(* IEC 61131-3 sources: SJ_AGV/PLC (part 2) *)

   END_STRUCT;
END_TYPE
TYPE
    LanSerialPort_T :
    STRUCT
        Protocol : DINT ;   (* Protocol used for IP communication.  *)
        IP : STRING ;   (* In case of Protocol set to UDP client or TCP client this should be set
to the IP address of the UDP/TCP server that the PLC connects to. With
Protocol set to UDP server or TCP server this specify the IP address of
the vehicle controller which clients should use.

In the case of Protocol set to UDP server or TCP server, the special
value "LAN" means that connections are only allowed on the
LAN interface and the special value "ANY" allows connections
on both the LAN interface and the WLAN interface.

Changing the address from the PLC will result in the connection being
closed. The new IP address will be used in the next PLC loop serial
read/write.  Note! It is not possible to change the address for a
range sensor connected using a LAN-serial-adapter.  *)
        Port : DINT ;   (* In case of Protocol set to UDP client or TCP client this should be set
to the port of the UDP/TCP server that the PLC connects to. With
Protocol set to UDP server or TCP server this specify the port on the
vehicle controller that the PLC opens for connections.

Changing the port from the PLC will result in the connection being
closed. The new port will be used in the next PLC loop serial
read/write.  Note! It is not possible to change the port for a range
sensor connected using a LAN-serial-adapter.  *)
        SendBuffer : BOOL ;   (* With SendBuffer set, outgoing data is sent over IP when the PLC
function block NDC_SERIAL_WRITE is called with argument
LENGTH=0. Without SendBuffer set, data is sent immediately but each IP
packet will contain at most 32 bytes data with more IP traffic as a
result.  *)

   END_STRUCT;
END_TYPE
TYPE
    UserDefined_T :
    STRUCT
        DoNavInit : BOOL ;   (* Boolean_1  *)
        Braker_Signal : BOOL ;   (* Boolean_2  *)
        DoLocalOrder : BOOL ;   (* Boolean_3  *)
        ChangeOrderMode : BOOL ;   (* Boolean_4  *)
        LowBatSim : BOOL ;   (* Boolean_5  *)
        Boolean_6 : BOOL ;   (* Boolean_6  *)
        Boolean_7 : BOOL ;   (* Boolean_7  *)
        Boolean_8 : BOOL ;   (* Boolean_8  *)
        Boolean_9 : BOOL ;   (* Boolean_9  *)
        Boolean_10_BlockPowOffEn : BOOL ;   (* Boolean_10  *)
        Boolean_11_LostPosPowOffEn : BOOL ;   (*   *)
        Boolean_12 : BOOL ;   (*   *)
        Boolean_13 : BOOL ;   (*   *)
        Boolean_14 : BOOL ;   (*   *)
        Boolean_15 : BOOL ;   (*   *)
        Boolean_16 : BOOL ;   (*   *)
        Boolean_17 : BOOL ;   (*   *)
        Boolean_18 : BOOL ;   (*   *)
        Boolean_19 : BOOL ;   (*   *)
        Boolean_20_OnlineOrderMode : BOOL ;   (* 1 = Local Mode; 0 = Host Mode  *)
        Boolean_21 : BOOL ;   (*   *)
        Boolean_22 : BOOL ;   (*   *)
        Boolean_23 : BOOL ;   (*   *)
        Boolean_24 : BOOL ;   (*   *)
        Boolean_25 : BOOL ;   (*   *)
        Boolean_26 : BOOL ;   (*   *)
        Boolean_27 : BOOL ;   (*   *)
        Boolean_28 : BOOL ;   (*   *)
        Boolean_29 : BOOL ;   (*   *)
        Boolean_30 : BOOL ;   (*   *)
        StopWord : DINT ;   (* Integer32_1  *)
        Integer32_2 : DINT ;   (* Integer32_2  *)
        Integer32_3 : DINT ;   (* Integer32_3  *)
        Integer32_4 : DINT ;   (* Integer32_4  *)
        Integer32_5 : DINT ;   (* Integer32_5  *)
        SlowDownDisable : DINT ;   (* Integer32_6  *)
        PPAEnable : DINT ;   (* Integer32_7  *)
        SafetyScannerTurnAngle : DINT ;   (* Integer32_8  *)
        NormalCreepDistance : DINT ;   (* Integer32_9  *)
        Integer32_10 : DINT ;   (* Integer32_10  *)
        Integer32_11 : DINT ;   (* Integer32_11  *)
        Integer32_12 : DINT ;   (* Integer32_12  *)
        Integer32_13 : DINT ;   (* Integer32_13  *)
        Integer32_14 : DINT ;   (* Integer32_14  *)
        Integer32_15 : DINT ;   (* Integer32_15  *)
        Integer32_16 : DINT ;   (* Integer32_16  *)
        Integer32_17 : DINT ;   (* Integer32_17  *)
        Integer32_18 : DINT ;   (* Integer32_18  *)
        Integer32_19 : DINT ;   (* Integer32_19  *)
        Integer32_20 : DINT ;   (* Integer32_20  *)
        Integer32_21 : DINT ;   (* Integer32_21  *)
        Integer32_22 : DINT ;   (* Integer32_22  *)
        Integer32_23 : DINT ;   (* Integer32_23  *)
        Integer32_24 : DINT ;   (* Integer32_24  *)
        Integer32_25 : DINT ;   (* Integer32_25  *)
        Integer32_26 : DINT ;   (* Integer32_26  *)
        Integer32_27 : DINT ;   (* Integer32_27  *)
        Integer32_28 : DINT ;   (* Integer32_28  *)
        Integer32_29 : DINT ;   (* Integer32_29  *)
        Integer32_30 : DINT ;   (* Integer32_30  *)
        Integer32_31 : DINT ;   (* Integer32_31  *)
        Integer32_32 : DINT ;   (* Integer32_32  *)
        Integer32_33 : DINT ;   (* Integer32_33  *)
        Integer32_34 : DINT ;   (* Integer32_34  *)
        Integer32_35 : DINT ;   (* Integer32_35  *)
        Integer32_36 : DINT ;   (* Integer32_36  *)
        Integer32_37 : DINT ;   (* Integer32_37  *)
        Integer32_38 : DINT ;   (* Integer32_38  *)
        Integer32_39 : DINT ;   (* Integer32_39  *)
        Integer32_40 : DINT ;   (* Integer32_40  *)
        Integer32_41 : DINT ;   (* Integer32_41  *)
        Integer32_42 : DINT ;   (* Integer32_42  *)
        Integer32_43 : DINT ;   (* Integer32_43  *)
        Integer32_44 : DINT ;   (* Integer32_44  *)
        Integer32_45 : DINT ;   (* Integer32_45  *)
        Integer32_46 : DINT ;   (* Integer32_46  *)
        Integer32_47 : DINT ;   (*   *)
        Integer32_48 : DINT ;   (*   *)
        Integer32_49 : DINT ;   (*   *)
        Integer32_50_BattLowVol : DINT ;   (*   *)
        Integer32_51_BattLowSel : DINT ;   (* 1=L or M or H, 2=M or H, 3=H  *)
        Integer32_52_PowOffTm : DINT ;   (* ms  *)
        Integer32_53 : DINT ;   (*   *)
        Integer32_54 : DINT ;   (*   *)
        Integer32_55_TravelDistance : DINT ;   (*   *)
        Integer32_56 : DINT ;   (*   *)
        Integer32_57 : DINT ;   (*   *)
        Integer32_58_LS2000_Attached_D : DINT ;   (*   *)
        Integer32_59_LS2000_Attached_H : DINT ;   (*   *)
        Integer32_60_LS2000_Attached_M : DINT ;   (*   *)

   END_STRUCT;
END_TYPE
TYPE
    SDIO_T :
    STRUCT
        IMUGyroX : INT ;   (* Gyroscope x-axis value, cdeg/s  *)
        IMUGyroY : INT ;   (* Gyroscope y-axis value, cdeg/s  *)
        IMUGyroZ : INT ;   (* Gyroscope z-axis value, cdeg/s  *)
        IMUAccX : INT ;   (* Accelerometer x-axis value, mg  *)
        IMUAccY : INT ;   (* Accelerometer x-axis value, mg  *)
        IMUAccZ : INT ;   (* Accelerometer x-axis value, mg  *)
        IMUError : UINT ;   (* IMU Error value  *)
        IMUGyroXScale : INT ;   (* Gyroscope x-axis scale value (the value 10000 corresponds to a real scale value of 1.0)  *)
        IMUGyroYScale : INT ;   (* Gyroscope y-axis scale value (the value 10000 corresponds to a real scale value of 1.0)  *)
        IMUGyroZScale : INT ;   (* Gyroscope z-axis scale value (the value 10000 corresponds to a real scale value of 1.0)  *)
        DigitalInput1_Polarity : BOOL ;   (* Digital Input 1 Polarity, pin #A22  *)
        DigitalInput2_Polarity : BOOL ;   (* Digital Input 2 Polarity, pin #A14  *)
        DigitalInput3_Polarity : BOOL ;   (* Digital Input 3 Polarity, pin #A7  *)
        DigitalInput4_Polarity : BOOL ;   (* Digital Input 4 Polarity, pin #A6  *)
        DigitalInput5_Polarity : BOOL ;   (* Digital Input 5 Polarity, pin #A13  *)
        DigitalInput6_Polarity : BOOL ;   (* Digital Input 6 Polarity, pin #A21  *)
        DigitalInput7_Polarity : BOOL ;   (* Digital Input 7 Polarity, pin #A20  *)
        DigitalInput8_Polarity : BOOL ;   (* Digital Input 8 Polarity, pin #A19  *)
        DigitalInput9_Polarity : BOOL ;   (* Digital Input 9 Polarity, pin #B22  *)
        DigitalInput10_Polarity : BOOL ;   (* Digital Input 10 Polarity, pin #B23  *)
        DigitalInput11_Polarity : BOOL ;   (* Digital Input 11 Polarity, pin #A18  *)
        DigitalInput12_Polarity : BOOL ;   (* Digital Input 12 Polarity, pin #A17  *)
        DigitalOutput2_Polarity : BOOL ;   (* Digital Output 2 Polarity, pin #B7  *)
        DigitalOutput3_Polarity : BOOL ;   (* Digital Output 3 Polarity, pin #B6  *)
        DigitalOutput4_Polarity : BOOL ;   (* Digital Output 4 Polarity, pin #B5  *)
        DigitalOutput5_Polarity : BOOL ;   (* Digital Output 5 Polarity, pin #B4  *)
        DigitalOutput6_Polarity : BOOL ;   (* Digital Output 6 Polarity, pin #B1  *)
        DigitalOutput7_Polarity : BOOL ;   (* Digital Output 7 Polarity, pin #B3  *)
        DigitalOutput8_Polarity : BOOL ;   (* Digital Output 8 Polarity, pin #B2  *)
        DigitalOutput12_Polarity : BOOL ;   (* Digital Output 12 Polarity, pin #A3  *)
        DigitalOutput13_Polarity : BOOL ;   (* Digital Output 13 Polarity, pin #A10  *)
        DigitalOutput14_Polarity : BOOL ;   (* Digital Output 14 Polarity, pin #A2  *)
        DigitalOutput15_Polarity : BOOL ;   (* Digital Output 15 Polarity, pin #A9  *)
        DigitalOutput16_Polarity : BOOL ;   (* Digital Output 16 Polarity, pin #A16  *)
        AnInp1_Scale : DINT ;   (* Analog Input 1 Scale, pin #B15  *)
        AnInp2_Scale : DINT ;   (* Analog Input 2 Scale, pin #B17  *)
        AnInp3_Scale : DINT ;   (* Analog Input 3 Scale, pin #B10  *)
        AnInp4_Scale : DINT ;   (* Analog Input 4 Scale, pin #B18  *)
        AnInp5_Scale : DINT ;   (* Analog Input 5 Scale, pin #B11  *)
        AnInp6_Scale : DINT ;   (* Analog Input 6 Scale, pin #B19  *)
        AnInp7_Scale : DINT ;   (* Analog Input 7 Scale, pin #B12  *)
        AnInp8_Scale : DINT ;   (* Analog Input 8 Scale, pin #B20  *)
        AnInp9_Scale : DINT ;   (* Analog Input 9 Scale, pin #B13  *)
        AnInp10_Scale : DINT ;   (* Analog Input 10 Scale, pin #B21  *)
        AnInp11_Scale : DINT ;   (* Analog Input 11 Scale, pin #B14  *)
        AnInp1_Delta : UDINT ;   (* Asynchroneous transmission will be triggered if input has changed more than this value since last transmission.  *)
        AnInp2_Delta : UDINT ;   (* Asynchroneous transmission will be triggered if input has changed more than this value since last transmission.  *)
        AnInp3_Delta : UDINT ;   (* Asynchroneous transmission will be triggered if input has changed more than this value since last transmission.  *)
        AnInp4_Delta : UDINT ;   (* Asynchroneous transmission will be triggered if input has changed more than this value since last transmission.  *)
        AnInp5_Delta : UDINT ;   (* Asynchroneous transmission will be triggered if input has changed more than this value since last transmission.  *)
        AnInp6_Delta : UDINT ;   (* Asynchroneous transmission will be triggered if input has changed more than this value since last transmission.  *)
        AnInp7_Delta : UDINT ;   (* Asynchroneous transmission will be triggered if input has changed more than this value since last transmission.  *)
        AnInp8_Delta : UDINT ;   (* Asynchroneous transmission will be triggered if input has changed more than this value since last transmission.  *)
        AnInp9_Delta : UDINT ;   (* Asynchroneous transmission will be triggered if input has changed more than this value since last transmission.  *)
        AnInp10_Delta : UDINT ;   (* Asynchroneous transmission will be triggered if input has changed more than this value since last transmission.  *)
        AnInp11_Delta : UDINT ;   (* Asynchroneous transmission will be triggered if input has changed more than this value since last transmission.  *)
        AnInp1_Offset : DINT ;   (* Analog Input 1 Offset, pin #B15  *)
        AnInp2_Offset : DINT ;   (* Analog Input 2 Offset, pin #B17  *)
        AnInp3_Offset : DINT ;   (* Analog Input 3 Offset, pin #B10  *)
        AnInp4_Offset : DINT ;   (* Analog Input 4 Offset, pin #B18  *)
        AnInp5_Offset : DINT ;   (* Analog Input 5 Offset, pin #B11  *)
        AnInp6_Offset : DINT ;   (* Analog Input 6 Offset, pin #B19  *)
        AnInp7_Offset : DINT ;   (* Analog Input 7 Offset, pin #B12  *)
        AnInp8_Offset : DINT ;   (* Analog Input 8 Offset, pin #B20  *)
        AnInp9_Offset : DINT ;   (* Analog Input 9 Offset, pin #B13  *)
        AnInp10_Offset : DINT ;   (* Analog Input 10 Offset, pin #B21  *)
        AnInp11_Offset : DINT ;   (* Analog Input 11 Offset, pin #B14  *)
        DigitalInput1_BTN_STR : BOOL ;   (* Digital Input 1 value, pin #A22  *)
        DigitalInput2_BTN_RST : BOOL ;   (* Digital Input 2 value, pin #A14  *)
        DigitalInput3_BMP_O1 : BOOL ;   (* Digital Input 3 value, pin #A7  *)
        DigitalInput4_BMP_O2 : BOOL ;   (* Digital Input 4 value, pin #A6  *)
        DigitalInput5_BTN_BRK : BOOL ;   (* Digital Input 5 value, pin #A13  *)
        DigitalInput6 : BOOL ;   (* Digital Input 6 value, pin #A21  *)
        DigitalInput7 : BOOL ;   (* Digital Input 7 value, pin #A20  *)
        DigitalInput8_BMP_E : BOOL ;   (* Digital Input 8 value, pin #A19  *)
        DigitalInput9 : BOOL ;   (* Digital Input 9 value, pin #B22  *)
        DigitalInput10 : BOOL ;   (* Digital Input 10 value, pin #B23  *)
        DigitalInput11 : BOOL ;   (* Digital Input 11 value, pin #A18  *)
        DigitalInput12_EMO : BOOL ;   (* Digital Input 12 value, pin #A17  *)
        AllOK_DigitalOutput1 : BOOL ;   (* Reserved Digital Output 1 (All-OK, pin #B8)  *)
        DigitalOutput2_LEDF_L : BOOL ;   (* Digital Output 2 value, pin #B7  *)
        DigitalOutput3_LEDF_R : BOOL ;   (* Digital Output 3 value, pin #B6  *)
        DigitalOutput4_LEDR_L : BOOL ;   (* Digital Output 4 value, pin #B5  *)
        DigitalOutput5_LEDR_R : BOOL ;   (* Digital Output 5 value, pin #B4  *)
        DigitalOutput6_LED_INPOS : BOOL ;   (* Digital Output 6 value, pin #B1  *)
        DigitalOutput7_LED_STR : BOOL ;   (* Digital Output 7 value, pin #B3  *)
        DigitalOutput8_LED_RST : BOOL ;   (* Digital Output 8 value, pin #B2  *)
        DigitalOutput12 : BOOL ;   (* Digital Output 12 value, pin #A3  *)
        DigitalOutput13_PWR_OFF : BOOL ;   (* Digital Output 13 value, pin #A10  *)
        DigitalOutput14_LED_BRK : BOOL ;   (* Digital Output 14 value, pin #A2  *)
        DigitalOutput15 : BOOL ;   (* Digital Output 15 value, pin #A9  *)
        DigitalOutput16_Charger : BOOL ;   (* Digital Output 16 value, pin #A16  *)
        AnalogInput1 : INT ;   (* Analog Input 1 value, pin #B15. The value is the applied input voltage (in Volts) * Scale + Offset  *)
        AnalogInput2 : INT ;   (* Analog Input 2 value, pin #B17. The value is the applied input voltage (in Volts) * Scale + Offset  *)
        AnalogInput3 : INT ;   (* Analog Input 3 value, pin #B10. The value is the applied input voltage (in Volts) * Scale + Offset  *)
        AnalogInput4 : INT ;   (* Analog Input 4 value, pin #B18. The value is the applied input voltage (in Volts) * Scale + Offset  *)
        AnalogInput5 : INT ;   (* Analog Input 5 value, pin #B11. The value is the applied input voltage (in Volts) * Scale + Offset  *)
        AnalogInput6 : INT ;   (* Analog Input 6 value, pin #B19. The value is the applied input voltage (in Volts) * Scale + Offset  *)
        AnalogInput7 : INT ;   (* Analog Input 7 value, pin #B12. The value is the applied input voltage (in Volts) * Scale + Offset  *)
        AnalogInput8 : INT ;   (* Analog Input 8 value, pin #B20. The value is the applied input voltage (in Volts) * Scale + Offset  *)
        AnalogInput9 : INT ;   (* Analog Input 9 value, pin #B13. The value is the applied input voltage (in Volts) * Scale + Offset  *)
        AnalogInput10 : INT ;   (* Analog Input 10 value, pin #B21. The value is the applied input voltage (in Volts) * Scale + Offset  *)
        AnalogInput11 : INT ;   (* Analog Input 11 value, pin #B14. The value is the applied input voltage (in Volts) * Scale + Offset  *)
        PWMOutput1 : INT ;   (* PWM Output 1 value, pin #A5. The value is the duty cycle of the output.  *)
        PWMOutput2 : INT ;   (* PWM Output 2 value, pin #A12. The value is the duty cycle of the output.  *)
        PWMOutput3 : INT ;   (* PWM Output 3 value, pin #A11. The value is the duty cycle of the output.  *)
        Reg1Output : INT ;   (* Regulator 1 output value  *)
        Reg2Output : INT ;   (* Regulator 2 output value  *)
        GroundFaultEvent : BOOL ;   (* If set to true, a ground fault will cause a system event 229.  *)
        GroundFaultActive : BOOL ;   (* True if a ground fault is present  *)
        Temperature : DINT ;   (* Current temperature  *)
        XV_Out : DINT ;   (* Current xv out voltage  *)
        B_Plus : DINT ;   (* Current b plus voltage  *)
        BusID : DINT ;   (* CAN bus ID  *)
        NodeID : DINT ;   (* CAN node ID  *)
        FailureAction : DINT ;   (* 0 = Background, the background programs takes action when an error occur in the device. 1 = PLC, no action from background program. The error should be handled by the PLC application.  *)
        ActiveInSafeState : BOOL ;   (* Decides if the device will start up in safe state.  *)
        NMTState : UDINT ;   (* The current CANopen state of the device.  *)
        SdoBufferSize : DINT ;   (* The current size of the client SDO buffer (read/write SDO's from the vehicle controller to this device).  *)
        IMUAxis : STRING ;   (* The axis in the IMU that gives the angular rate for vehicle.  *)
        IMUNavActive : BOOL ;   (* Use the angular rate from the IMU when calculating the position of the vehicle.  *)

   END_STRUCT;
END_TYPE
TYPE
    CAN_IO_3_T :
    STRUCT
        DigitalInput1_SteerLimitF_L : BOOL ;   (* Digital Input 1 value  *)
        DigitalInput2_SteerLimitF_R : BOOL ;   (* Digital Input 2 value  *)
        DigitalInput3_SteerLimitR_L : BOOL ;   (* Digital Input 3 value  *)
        DigitalInput4_SteerLimitR_R : BOOL ;   (* Digital Input 4 value  *)
        DigitalInput5_LIMF_O : BOOL ;   (* Digital Input 5 value  *)
        DigitalInput6_LIMR_O : BOOL ;   (* Digital Input 6 value  *)
        DigitalInput7 : BOOL ;   (* Digital Input 7 value  *)
        DigitalInput8 : BOOL ;   (* Digital Input 8 value  *)
        DigitalInput9_AreaF_IN1 : BOOL ;   (* Digital Input 9 value  *)
        DigitalInput10_AreaF_IN2 : BOOL ;   (* Digital Input 10 value  *)
        DigitalInput11 : BOOL ;   (* Digital Input 11 value  *)
        DigitalInput12 : BOOL ;   (* Digital Input 12 value  *)
        DigitalInput13_AreaR_IN1 : BOOL ;   (* Digital Input 13 value  *)
        DigitalInput14_AreaR_IN2 : BOOL ;   (* Digital Input 14 value  *)
        DigitalInput15 : BOOL ;   (* Digital Input 15 value  *)
        DigitalInput16 : BOOL ;   (* Digital Input 16 value  *)
        DigitalOutput1_BuzzerCh1 : BOOL ;   (* Digital Output 1 value  *)
        DigitalOutput2_BuzzerCh2 : BOOL ;   (* Digital Output 2 value  *)
        DigitalOutput3_BuzzerCh3 : BOOL ;   (* Digital Output 3 value  *)
        DigitalOutput4_BuzzerCh4 : BOOL ;   (* Digital Output 4 value  *)
        DigitalOutput5 : BOOL ;   (* Digital Output 5 value  *)
        DigitalOutput6 : BOOL ;   (* Digital Output 6 value  *)
        DigitalOutput7 : BOOL ;   (* Digital Output 7 value  *)
        DigitalOutput8 : BOOL ;   (* Digital Output 8 value  *)
        DigitalOutput9_AreaF_SW1 : BOOL ;   (* Digital Output 9 value  *)
        DigitalOutput10_AreaF_SW2 : BOOL ;   (* Digital Output 10 value  *)
        DigitalOutput11 : BOOL ;   (* Digital Output 11 value  *)
        DigitalOutput12 : BOOL ;   (* Digital Output 12 value  *)
        DigitalOutput13_AreaR_SW1 : BOOL ;   (* Digital Output 13 value  *)
        DigitalOutput14_AreaR_SW2 : BOOL ;   (* Digital Output 14 value  *)
        DigitalOutput15 : BOOL ;   (* Digital Output 15 value  *)
        DigitalOutput16 : BOOL ;   (* Digital Output 16 value  *)
        BusID : DINT ;   (* CAN bus ID  *)
        NodeID : DINT ;   (* CAN node ID  *)
        FailureAction : DINT ;   (* 0 = Background, the background programs takes action when an error occur in the device. 1 = PLC, no action from background program. The error should be handled by the PLC application.  *)
        ActiveInSafeState : BOOL ;   (* Decides if the device will start up in safe state.  *)
        NMTState : UDINT ;   (* The current CANopen state of the device.  *)
        SdoBufferSize : DINT ;   (* The current size of the client SDO buffer (read/write SDO's from the vehicle controller to this device).  *)

   END_STRUCT;
END_TYPE
TYPE
    DCD_5_T :
    STRUCT
        MotorCurrentRegP : INT ;   (* Motor Parameter: Proportional gain in the PI-parts of the current controller.  *)
        MotorCurrentRegI : INT ;   (* Motor Parameter: Integral gain in the PI-parts of the current controller.  *)
        MaxCommandSpeed : UINT ;   (* Max command speed  *)
        ForwardMaxAccTorqueCurrent : INT ;   (* Maximum allowed torque current during forward acceleration.  *)
        ReverseMaxAccTorqueCurrent : INT ;   (* Maximum allowed torque current during reverse acceleration.  *)
        MaxTorqueCurrentChange : INT ;   (* The maximum allowed change during 1 ms (i.e. derivate) of the Torque Current that is allowed. A too high derivate may for example introduce noise in the gear.  *)
        ForwardMaxBrakeTorqueCurrent : INT ;   (* Maximum allowed torque current during forward braking/deceleration.  *)
        ReverseMaxBrakeTorqueCurrent : INT ;   (* Maximum allowed torque current during reverse braking/deceleration.  *)
        SpeedRegP : UINT ;   (* Proportional gain in the PI-parts of the speed controller.  *)
        SpeedRegI : UINT ;   (* Integral gain in the PI-parts of the speed controller.  *)
        RegSupervisionCheckOutHysteresis : UINT ;   (* Current limit for supervision. Supervision is enabled when the requested torque current goes above this limit. (Regulator supervision 0x6210)  *)
        RegSupervisionFailureDelay : UINT ;   (* Delay before safe state in absence of movement in correct direction. 0 = Disable. (Regulator supervision 0x6210)  *)
        ReverseEncoderDirection : BOOL ;   (* Set true to reverse encoder direction. Same effect as swapping A and B signals.  *)
        VoltageFeedback : BOOL ;   (* Set true to use motor voltage as speed feedback instead of encoder. (Speed scale: 1024 = 48 V)  *)
        SpeedRegOffset : INT ;   (* Current to compensate for friction. Added to speed regulator output with sign depending on the command speed.  *)
        ReadyToSwitchOn : BOOL ;   (* Ready To Switch On (Dc bus is charged)  *)
        SwitchedOn : BOOL ;   (* Switched On  *)
        PowerStageEnabled : BOOL ;   (* Power Stage Enabled  *)
        Error : BOOL ;   (* Error  *)
        SwitchOnDisabled : BOOL ;   (* Switch On Disabled	(Dc bus voltage to low, charging timeout)  *)
        Warning : BOOL ;   (* Warning  *)
        DriveEncScale : UDINT ;   (* The number of pulses per 1000 mm.  *)
        DriveEncDist : UINT ;   (* Drive Encoder Distance  *)
        DriveEncSpeed : INT ;   (* Drive Enc Speed  *)
        DigitalInput2_OverRelayFS : BOOL ;   (* Digital Input 2 value, pin 14  *)
        DigitalInput3_OverRelayFD : BOOL ;   (* Digital Input 3 value, pin 13  *)
        SwitchOn : BOOL ;   (* Switch On  *)
        EnablePowerStage : BOOL ;   (* Enable Power Stage  *)
        SetSpeed : INT ;   (* Set Speed  *)
        AllOK_DigitalOutput1 : BOOL ;   (* Reserved Digital Output 1 value, pin 2  *)
        DigitalOutput2_Braker : BOOL ;   (* Digital Output 2 value, pin 18  *)
        DigitalOutput3 : BOOL ;   (* Digital Output 3 value, pin 21  *)
        DigitalOutput4 : BOOL ;   (* Digital Output 4 value, pin 22  *)
        DcBusVoltage : UINT ;   (* Runtime voltage measurement on the B+ input  *)
        TorqueCurrentReference : INT ;   (* Output from speed controller, input to current controller.  *)
        TorqueCurrent : INT ;   (* Actual torque current in current controller.  *)
        HeatsinkTemperature : INT ;   (* Temperature of the heatsink  *)
        ExtendedWarnings : UDINT ;   (* Extended Warnings set by the drive, valid when Warning bit is set  *)
        ExtendedErrors : UDINT ;   (* Extended Errors set by the drive, valid when Error bit is set  *)
        RegSupervisionTimer : UINT ;   (* Timer counting absence of movement in correct direction. See: Reg Supervision Failure Delay  *)
        RegSupervisionTimerMax : UINT ;   (* Max value of Reg Supervision Timer since power on.  *)
        BusID : DINT ;   (* CAN bus ID  *)
        NodeID : DINT ;   (* CAN node ID  *)
        FailureAction : DINT ;   (* 0 = Background, the background programs takes action when an error occur in the device. 1 = PLC, no action from background program. The error should be handled by the PLC application.  *)
        ActiveInSafeState : BOOL ;   (* Decides if the device will start up in safe state.  *)
        NMTState : UDINT ;   (* The current CANopen state of the device.  *)
        SdoBufferSize : DINT ;   (* The current size of the client SDO buffer (read/write SDO's from the vehicle controller to this device).  *)

   END_STRUCT;
END_TYPE
TYPE
    DCD_6_T :
    STRUCT
        MotorCurrentRegP : INT ;   (* Motor Parameter: Proportional gain in the PI-parts of the current controller.  *)
        MotorCurrentRegI : INT ;   (* Motor Parameter: Integral gain in the PI-parts of the current controller.  *)
        ForwardMaxAccTorqueCurrent : INT ;   (* Maximum allowed torque current during forward acceleration.  *)
        ReverseMaxAccTorqueCurrent : INT ;   (* Maximum allowed torque current during reverse acceleration.  *)
        MaxTorqueCurrentChange : INT ;   (* The maximum allowed change during 1 ms (i.e. derivate) of the Torque Current that is allowed. A too high derivate may for example introduce noise in the gear.  *)
        ForwardMaxBrakeTorqueCurrent : INT ;   (* Maximum allowed torque current during forward braking/deceleration.  *)
        ReverseMaxBrakeTorqueCurrent : INT ;   (* Maximum allowed torque current during reverse braking/deceleration.  *)
        SpeedRegP : UINT ;   (* Proportional gain in the PI-parts of the speed controller.  *)
        SpeedRegI : UINT ;   (* Integral gain in the PI-parts of the speed controller.  *)
        RegSupervisionCheckOutHysteresis : UINT ;   (* Current limit for supervision. Supervision is enabled when the requested torque current goes above this limit. (Regulator supervision 0x6210)  *)
        RegSupervisionFailureDelay : UINT ;   (* Delay before safe state in absence of movement in correct direction. 0 = Disable. (Regulator supervision 0x6210)  *)
        SteerEncScale : UDINT ;   (* Steering Encoder Scale  *)
        SteerEncOffset : INT ;   (* Steering Encoder Offset (Position of Sync pulse)  *)
        PosRegP : INT ;   (* Proportional gain in the PI-parts of the position controller.  *)
        PosRegI : INT ;   (* Integral gain in the PI-parts of the position controller.  *)
        LimOutMax : INT ;   (* Max motor speed as output from position controller and input to speed controller.
VoltageFeedback: 1024 = 48V, Otherwise: 16384 = 90 deg/s  *)
        MaxWheelAngle : INT ;   (* Wheel Angle Limit. 0 = No Limit  *)
        SlowDownZone : INT ;   (* Speed limited zone approaching MaxWheelAngle.  *)
        LimOutMaxSlowDownZone : UINT ;   (* Speed limit for the slow down zone.  *)
        EndLimitSwitchPolarity : UINT ;   (* Polarity of end limit switch. Default is active high.  *)
        SyncGate : BOOL ;   (* Set true to allow sync. Set to false to reject unwanted sync pulse in multi turn application.  *)
        SyncFilter : UINT ;   (* Window where we expect sync pulse to appear  *)
        SyncEmergency : BOOL ;   (* Encoder Sync Emergency. 0 = Sync Emergency disabled. OBS! Disabling the sync emergency can be a serious safety issue!  *)
        ReverseEncoderDirection : BOOL ;   (* Set true to reverse encoder direction. Same effect as swapping A and B signals.  *)
        VoltageFeedback : BOOL ;   (* Set true to use motor voltage as speed feedback instead of encoder. (Speed scale: 1024 = 48 V)  *)
        SpeedRegOffset : INT ;   (* Current to compensate for friction. Added to speed regulator output with sign depending on the command speed.  *)
        ReadyToSwitchOn : BOOL ;   (* Ready To Switch On (Dc bus is charged)  *)
        SwitchedOn : BOOL ;   (* Switched On  *)
        PowerStageEnabled : BOOL ;   (* Power Stage Enabled  *)
        Error : BOOL ;   (* Error  *)
        SwitchOnDisabled : BOOL ;   (* Switch On Disabled	(Dc bus voltage to low, charging timeout)  *)
        Warning : BOOL ;   (* Warning  *)
        WheelAngle : INT ;   (* Wheel Angle  *)
        Reserved_DigitalInput2 : BOOL ;   (* Digital Input 2 value, encoder sync, pin 14  *)
        Reserved_DigitalInput3 : BOOL ;   (* Digital Input 3 value, end limit switch, pin 13  *)
        SwitchOn : BOOL ;   (* Switch On  *)
        EnablePowerStage : BOOL ;   (* Enable Power Stage  *)
        SetAngle : INT ;   (* Set Angle  *)
        DigitalOutput1 : BOOL ;   (* Digital Output 1 value, pin 2  *)
        DigitalOutput2 : BOOL ;   (* Digital Output 2 value, pin 18  *)
        DigitalOutput3 : BOOL ;   (* Digital Output 3 value, pin 21  *)
        DigitalOutput4 : BOOL ;   (* Digital Output 4 value, pin 22  *)
        DcBusVoltage : UINT ;   (* Runtime voltage measurement on the B+ input  *)
        TorqueCurrentReference : INT ;   (* Output from speed controller, input to current controller.  *)
        TorqueCurrent : INT ;   (* Actual torque current in current controller.  *)
        EncoderStatus : UINT ;   (* Bit0 - Sync Valid. Set when first sync pulse inside the sync window has been detected  *)
        EncoderCounterValue : UINT ;   (* Number of pulse edges captured.  *)
        SpuriousSyncCounter : UINT ;   (* Counter for sync pulses detected outside sync window. Valid after first sync pulse inside the sync window has been detected  *)
        MissingSyncCounter : UINT ;   (* Counter for expected but not present sync pulses inside sync window. Valid after first sync pulse inside the sync window has been detected  *)
        HeatsinkTemperature : INT ;   (* Temperature of the heatsink  *)
        ExtendedWarnings : UDINT ;   (* Extended Warnings set by the drive, valid when Warning bit is set  *)
        ExtendedErrors : UDINT ;   (* Extended Errors set by the drive, valid when Error bit is set  *)
        RegSupervisionTimer : UINT ;   (* Timer counting absence of movement in correct direction. See: Reg Supervision Failure Delay  *)
        RegSupervisionTimerMax : UINT ;   (* Max value of Reg Supervision Timer since power on.  *)
        BusID : DINT ;   (* CAN bus ID  *)
        NodeID : DINT ;   (* CAN node ID  *)
        FailureAction : DINT ;   (* 0 = Background, the background programs takes action when an error occur in the device. 1 = PLC, no action from background program. The error should be handled by the PLC application.  *)
        ActiveInSafeState : BOOL ;   (* Decides if the device will start up in safe state.  *)
        NMTState : UDINT ;   (* The current CANopen state of the device.  *)
        SdoBufferSize : DINT ;   (* The current size of the client SDO buffer (read/write SDO's from the vehicle controller to this device).  *)

   END_STRUCT;
END_TYPE
TYPE
    DCD_7_T :
    STRUCT
        MotorCurrentRegP : INT ;   (* Motor Parameter: Proportional gain in the PI-parts of the current controller.  *)
        MotorCurrentRegI : INT ;   (* Motor Parameter: Integral gain in the PI-parts of the current controller.  *)
        MaxCommandSpeed : UINT ;   (* Max command speed  *)
        ForwardMaxAccTorqueCurrent : INT ;   (* Maximum allowed torque current during forward acceleration.  *)
        ReverseMaxAccTorqueCurrent : INT ;   (* Maximum allowed torque current during reverse acceleration.  *)
        MaxTorqueCurrentChange : INT ;   (* The maximum allowed change during 1 ms (i.e. derivate) of the Torque Current that is allowed. A too high derivate may for example introduce noise in the gear.  *)
        ForwardMaxBrakeTorqueCurrent : INT ;   (* Maximum allowed torque current during forward braking/deceleration.  *)
        ReverseMaxBrakeTorqueCurrent : INT ;   (* Maximum allowed torque current during reverse braking/deceleration.  *)
        SpeedRegP : UINT ;   (* Proportional gain in the PI-parts of the speed controller.  *)
        SpeedRegI : UINT ;   (* Integral gain in the PI-parts of the speed controller.  *)
        RegSupervisionCheckOutHysteresis : UINT ;   (* Current limit for supervision. Supervision is enabled when the requested torque current goes above this limit. (Regulator supervision 0x6210)  *)
        RegSupervisionFailureDelay : UINT ;   (* Delay before safe state in absence of movement in correct direction. 0 = Disable. (Regulator supervision 0x6210)  *)
        ReverseEncoderDirection : BOOL ;   (* Set true to reverse encoder direction. Same effect as swapping A and B signals.  *)
        VoltageFeedback : BOOL ;   (* Set true to use motor voltage as speed feedback instead of encoder. (Speed scale: 1024 = 48 V)  *)
        SpeedRegOffset : INT ;   (* Current to compensate for friction. Added to speed regulator output with sign depending on the command speed.  *)
        ReadyToSwitchOn : BOOL ;   (* Ready To Switch On (Dc bus is charged)  *)
        SwitchedOn : BOOL ;   (* Switched On  *)
        PowerStageEnabled : BOOL ;   (* Power Stage Enabled  *)
        Error : BOOL ;   (* Error  *)
        SwitchOnDisabled : BOOL ;   (* Switch On Disabled	(Dc bus voltage to low, charging timeout)  *)
        Warning : BOOL ;   (* Warning  *)
        DriveEncScale : UDINT ;   (* The number of pulses per 1000 mm.  *)
        DriveEncDist : UINT ;   (* Drive Encoder Distance  *)
        DriveEncSpeed : INT ;   (* Drive Enc Speed  *)
        DigitalInput2_OverRelayRS : BOOL ;   (* Digital Input 2 value, pin 14  *)
        DigitalInput3_OverRelayRD : BOOL ;   (* Digital Input 3 value, pin 13  *)
        SwitchOn : BOOL ;   (* Switch On  *)
        EnablePowerStage : BOOL ;   (* Enable Power Stage  *)
        SetSpeed : INT ;   (* Set Speed  *)
        DigitalOutput1 : BOOL ;   (* Digital Output 1 value, pin 2  *)
        DigitalOutput2_Braker : BOOL ;   (* Digital Output 2 value, pin 18  *)
        DigitalOutput3 : BOOL ;   (* Digital Output 3 value, pin 21  *)
        DigitalOutput4 : BOOL ;   (* Digital Output 4 value, pin 22  *)
        DcBusVoltage : UINT ;   (* Runtime voltage measurement on the B+ input  *)
        TorqueCurrentReference : INT ;   (* Output from speed controller, input to current controller.  *)
        TorqueCurrent : INT ;   (* Actual torque current in current controller.  *)
        HeatsinkTemperature : INT ;   (* Temperature of the heatsink  *)
        ExtendedWarnings : UDINT ;   (* Extended Warnings set by the drive, valid when Warning bit is set  *)
        ExtendedErrors : UDINT ;   (* Extended Errors set by the drive, valid when Error bit is set  *)
        RegSupervisionTimer : UINT ;   (* Timer counting absence of movement in correct direction. See: Reg Supervision Failure Delay  *)
        RegSupervisionTimerMax : UINT ;   (* Max value of Reg Supervision Timer since power on.  *)
        BusID : DINT ;   (* CAN bus ID  *)
        NodeID : DINT ;   (* CAN node ID  *)
        FailureAction : DINT ;   (* 0 = Background, the background programs takes action when an error occur in the device. 1 = PLC, no action from background program. The error should be handled by the PLC application.  *)
        ActiveInSafeState : BOOL ;   (* Decides if the device will start up in safe state.  *)
        NMTState : UDINT ;   (* The current CANopen state of the device.  *)
        SdoBufferSize : DINT ;   (* The current size of the client SDO buffer (read/write SDO's from the vehicle controller to this device).  *)

   END_STRUCT;
END_TYPE
TYPE
    DCD_8_T :
    STRUCT
        MotorCurrentRegP : INT ;   (* Motor Parameter: Proportional gain in the PI-parts of the current controller.  *)
        MotorCurrentRegI : INT ;   (* Motor Parameter: Integral gain in the PI-parts of the current controller.  *)
        ForwardMaxAccTorqueCurrent : INT ;   (* Maximum allowed torque current during forward acceleration.  *)
        ReverseMaxAccTorqueCurrent : INT ;   (* Maximum allowed torque current during reverse acceleration.  *)
        MaxTorqueCurrentChange : INT ;   (* The maximum allowed change during 1 ms (i.e. derivate) of the Torque Current that is allowed. A too high derivate may for example introduce noise in the gear.  *)
        ForwardMaxBrakeTorqueCurrent : INT ;   (* Maximum allowed torque current during forward braking/deceleration.  *)
        ReverseMaxBrakeTorqueCurrent : INT ;   (* Maximum allowed torque current during reverse braking/deceleration.  *)
        SpeedRegP : UINT ;   (* Proportional gain in the PI-parts of the speed controller.  *)
        SpeedRegI : UINT ;   (* Integral gain in the PI-parts of the speed controller.  *)
        RegSupervisionCheckOutHysteresis : UINT ;   (* Current limit for supervision. Supervision is enabled when the requested torque current goes above this limit. (Regulator supervision 0x6210)  *)
        RegSupervisionFailureDelay : UINT ;   (* Delay before safe state in absence of movement in correct direction. 0 = Disable. (Regulator supervision 0x6210)  *)
        SteerEncScale : UDINT ;   (* Steering Encoder Scale  *)
        SteerEncOffset : INT ;   (* Steering Encoder Offset (Position of Sync pulse)  *)
        PosRegP : INT ;   (* Proportional gain in the PI-parts of the position controller.  *)
        PosRegI : INT ;   (* Integral gain in the PI-parts of the position controller.  *)
        LimOutMax : INT ;   (* Max motor speed as output from position controller and input to speed controller.
VoltageFeedback: 1024 = 48V, Otherwise: 16384 = 90 deg/s  *)
        MaxWheelAngle : INT ;   (* Wheel Angle Limit. 0 = No Limit  *)
        SlowDownZone : INT ;   (* Speed limited zone approaching MaxWheelAngle.  *)
        LimOutMaxSlowDownZone : UINT ;   (* Speed limit for the slow down zone.  *)
        EndLimitSwitchPolarity : UINT ;   (* Polarity of end limit switch. Default is active high.  *)
        SyncGate : BOOL ;   (* Set true to allow sync. Set to false to reject unwanted sync pulse in multi turn application.  *)
        SyncFilter : UINT ;   (* Window where we expect sync pulse to appear  *)
        SyncEmergency : BOOL ;   (* Encoder Sync Emergency. 0 = Sync Emergency disabled. OBS! Disabling the sync emergency can be a serious safety issue!  *)
        ReverseEncoderDirection : BOOL ;   (* Set true to reverse encoder direction. Same effect as swapping A and B signals.  *)
        VoltageFeedback : BOOL ;   (* Set true to use motor voltage as speed feedback instead of encoder. (Speed scale: 1024 = 48 V)  *)
        SpeedRegOffset : INT ;   (* Current to compensate for friction. Added to speed regulator output with sign depending on the command speed.  *)
        ReadyToSwitchOn : BOOL ;   (* Ready To Switch On (Dc bus is charged)  *)
        SwitchedOn : BOOL ;   (* Switched On  *)
        PowerStageEnabled : BOOL ;   (* Power Stage Enabled  *)
        Error : BOOL ;   (* Error  *)
        SwitchOnDisabled : BOOL ;   (* Switch On Disabled	(Dc bus voltage to low, charging timeout)  *)
        Warning : BOOL ;   (* Warning  *)
        WheelAngle : INT ;   (* Wheel Angle  *)
        Reserved_DigitalInput2 : BOOL ;   (* Digital Input 2 value, encoder sync, pin 14  *)
        Reserved_DigitalInput3 : BOOL ;   (* Digital Input 3 value, end limit switch, pin 13  *)
        SwitchOn : BOOL ;   (* Switch On  *)
        EnablePowerStage : BOOL ;   (* Enable Power Stage  *)
        SetAngle : INT ;   (* Set Angle  *)
        DigitalOutput1 : BOOL ;   (* Digital Output 1 value, pin 2  *)
        DigitalOutput2 : BOOL ;   (* Digital Output 2 value, pin 18  *)
        DigitalOutput3 : BOOL ;   (* Digital Output 3 value, pin 21  *)
        DigitalOutput4 : BOOL ;   (* Digital Output 4 value, pin 22  *)
        DcBusVoltage : UINT ;   (* Runtime voltage measurement on the B+ input  *)
        TorqueCurrentReference : INT ;   (* Output from speed controller, input to current controller.  *)
        TorqueCurrent : INT ;   (* Actual torque current in current controller.  *)
        EncoderStatus : UINT ;   (* Bit0 - Sync Valid. Set when first sync pulse inside the sync window has been detected  *)
        EncoderCounterValue : UINT ;   (* Number of pulse edges captured.  *)
        SpuriousSyncCounter : UINT ;   (* Counter for sync pulses detected outside sync window. Valid after first sync pulse inside the sync window has been detected  *)
        MissingSyncCounter : UINT ;   (* Counter for expected but not present sync pulses inside sync window. Valid after first sync pulse inside the sync window has been detected  *)
        HeatsinkTemperature : INT ;   (* Temperature of the heatsink  *)
        ExtendedWarnings : UDINT ;   (* Extended Warnings set by the drive, valid when Warning bit is set  *)
        ExtendedErrors : UDINT ;   (* Extended Errors set by the drive, valid when Error bit is set  *)
        RegSupervisionTimer : UINT ;   (* Timer counting absence of movement in correct direction. See: Reg Supervision Failure Delay  *)
        RegSupervisionTimerMax : UINT ;   (* Max value of Reg Supervision Timer since power on.  *)
        BusID : DINT ;   (* CAN bus ID  *)
        NodeID : DINT ;   (* CAN node ID  *)
        FailureAction : DINT ;   (* 0 = Background, the background programs takes action when an error occur in the device. 1 = PLC, no action from background program. The error should be handled by the PLC application.  *)
        ActiveInSafeState : BOOL ;   (* Decides if the device will start up in safe state.  *)
        NMTState : UDINT ;   (* The current CANopen state of the device.  *)
        SdoBufferSize : DINT ;   (* The current size of the client SDO buffer (read/write SDO's from the vehicle controller to this device).  *)

   END_STRUCT;
END_TYPE

TYPE
    NDC8_T :
    STRUCT
	NavInit : NavInit_T;
	    Mcd : MCD7P_T;
	    Position : Position_T;
	    Guidance : Guidance_T;
	    Autoinsert : Autoinsert_T;
	    Opt : GenericDisplay_T;
	    LayoutPosition : LayoutPosition_T;
	    Automatic : Automatic_T;
	    Manual : Manual_T;
	    BlackBox : BlackBox_T;
	    LocalOrder : LocalOrder_T;
	    SSIO : SSIO_T;
	    SegmentTrigger : SegmentTrigger_T;
	    PointTrigger : PointTrigger_T;
	    LoadDocking : LoadDocking_T;
	    LoadOperation : LoadOperation_T;
	    CANBus1 : CANBus_T;
	    CANBus2 : CANBus_T;
	    VehicleControl : VehicleControl_T;
	    VehicleOptions : VehicleOptions_T;
	    PLC_Application : PLC_Application_T;
	    COM1 : SerialPort_RS232_T;
	    COM2 : SerialPort_RS422_T;
	    COM3 : SerialPort_RS485_T;
	    Master : Master_T;
	    Vmc : Vmc_T;
	    Wlan : Wlan_T;
	    OMPLC : OMPLC_T;
	    VehicleApplication : VehicleApplication_T;
	    Layout : Layout_T;
	    CanOpenMaster : CanOpenMaster_T;
	    CanOpenEmergency : CanOpenEmergency_T;
	    PLCEmergency : PLCEmergency_T;
	    SlavebusControl : SlavebusControl_T;
	    UserDefined : UserDefined_T;
	    ExternalPath : ExternalPath_T;
	    BlockedInfo : BlockedInfo_T;
	    FrontWheel : WheelSD_T;
	    RearWheel : WheelSD_T;
	    COM5 : LanSerialPort_T;
	    LS2000 : LS2000Scanner_T;
	    Vehicle : Vehicle_T;
	    ReflectorInit : ReflectorInit_T;
	    NaturalNavigator : NaturalNavigator_T;
	    VehicleNavigator : VehicleNavigator_T;
	    ReflectorNavigator : ReflectorNavigator_T;
	    COM6 : LanSerialPort_T;
	    COM7 : LanSerialPort_T;
	    DCD_5 : DCD_5_T;
	    DCD_6 : DCD_6_T;
	    DCD_7 : DCD_7_T;
	    DCD_8 : DCD_8_T;
	    SDIO : SDIO_T;
	    CAN_IO_3 : CAN_IO_3_T;

   END_STRUCT;
END_TYPE

(* ---- USERTYPE.TYP ---- *)
[IEC_IEC_NORM]
TYPE

END_TYPE

(* ---- INPUTMAP_FB.ST ---- *)
FUNCTION_BLOCK INPUTMAP_FB
VAR_EXTERNAL
NDC8:NDC8_T;
Input : Input_T;

END_VAR

VAR_INPUT

END_VAR

VAR_OUTPUT

END_VAR

VAR
	StartSwitchRise : R_Trig;
	StartSwitchFlag : BOOL;
	StartDelay : TON;
	McdAutoR : R_Trig;
	McdAutoFlag : BOOL;
	OrderMode:OrderMode_FB;
END_VAR
(*
------------------------------------------------------------------------------------
 Input_Map_FB
 -----------

 Description:
	 Used to map actual inputs to generic variables.

-------------------------------------------------------------------------------------*)

(* Minimum required inputs * )
INPUT.ForkEncSyncValid		:= NDC8.. ;
								:= TRUE; 									if using CAN encoder or analog input.

INPUT.SteerEncSyncValid		:= NDC8.. ;
								:= (NDC8.DCD_5.EncoderStatus = 1);			for DCD
								:= TRUE ;									for ACD with CAN encoder
								:= NDC8.SDIO.Enc1SyncValid ;				for ACD with incremental encoder

( * Frequently used inputs  * )
INPUT.Reset_PB				:= NDC8.. ;
INPUT.SafetyScannerStop1	:= NDC8.. ;
INPUT.SafetyScannerStop2	:= NDC8.. ;
INPUT.LoadOnBoard			:= NDC8.. ;
INPUT.TractionSpeed			:= NDC8.. ;		( * DINT * )
INPUT.TractionDistance		:= NDC8.. ;		( * INT * )
INPUT.SafetyScannerSlowDown	:= NDC8.. ;

Input.ManualForkUp_PB 		:= NDC8.MCD.Button8;	( * MCD Load up.	Move the fork up. * )
Input.ManualForkDown_PB 	:= NDC8.MCD.Button9;	( * MCD Load down.	Move the fork down. * )
Input.ZeroSteerAngle_PB		:= NDC8.MCD.Button11;   ( * MCD Load right. Set the steerangle to zero in manual mode * )
Input.ChangeSteerMode_PB	:= NDC8.MCD.Button10;	( * MCD Load left. 	Switch steer modes in manual or semi (QUAD) * )

Input.LowBattery			:= NDC8.SDIO.B_Plus < 2200 ;			( * Simple example of battery level supervision.
								Normally CVC600 is connected via filter or DC/DC Battery+, so this value is not valid. * )
Input.BatteryLevel			:=    ( * INT * )

Input.SteerEncAngle			:= NDC8.. ;		( * DINT * )
								:= INT_to_DINT(NDC8.DCD_6.WheelAngle) ;  	for DCD
								:= NDC8.CAN_Enc_x.SteerEncAngle ;			for ACD with CAN encoder
								:= INT_TO_DINT(NDC8.SDIO.Enc1Angle) ;		for ACD with incremental encoder
NDC8.xCD_x.SyncGate			:= NDC..										for ACD or DCD with multi turn incremental steer encoder.

Input.ForkSpeed					:= NDC8.. ;		( * DINT * )
INPUT.ForkHeight				:= NDC8.. ;		( * DINT * )
INPUT.ForkTipSensorLeft			:= NDC8.. ;
INPUT.ForkTipSensorRight		:= NDC8.. ;
INPUT.ForkTipCentreLeft			:= NDC8.. ;
INPUT.ForkTipCentreRight		:= NDC8.. ;
INPUT.SideSensorRightBackward	:= NDC8.. ;
INPUT.SideSensorRightForward	:= NDC8.. ;
INPUT.SideSensorLeftBackward	:= NDC8.. ;
INPUT.SideSensorLeftForward		:= NDC8.. ;

*)

(* In the vehicle documentation, and the INPUTS.TYP, more examples of InputMap_FB is found. *)
;
(* Button *)
INPUT.Reset_PB := NDC8.SDIO.DigitalInput2_BTN_RST;

Input.ZeroSteerAngle_PB			:= 	NDC8.MCD.Button7;

INPUT.TractionSpeed := NDC8.VehicleControl.SetSpeed;

Input.ChangeSteerMode_PB	:= NDC8.MCD.Button10;
Input.ChangeSteerMode_PB2	:= NDC8.Mcd.Button11;

if NDC8.SDIO.DigitalInput3_BMP_O1 = TRUE or NDC8.SDIO.DigitalInput4_BMP_O2 = TRUE then
	StopSafety := TRUE;
else
	StopSafety := FALSE;
end_if;

StartSwitchRise(CLK:= NDC8.SDIO.DigitalInput1_BTN_STR);

if INPUT.StartMode = FALSE and StartSwitchRise.Q then
	INPUT.StartMode := TRUE;
elsif g_ErrorCode <> 0 and g_ErrorCode <> 155 and g_ErrorCode <> 156 then
	INPUT.StartMode := FALSE;
end_if;

if INPUT.Manual = TRUE then
	INPUT.StartMode := FALSE;
end_if;

McdAutoR(CLK := NDC8.Mcd.Button1);

if McdAutoR.Q then
	Input.BuzzerByPass := FALSE;
end_if;

if NDC8.DCD_6.EncoderStatus = 1 and NDC8.DCD_8.EncoderStatus = 1 then
	INPUT.SteerEncSyncValid := TRUE;
else
	INPUT.SteerEncSyncValid := FALSE;
end_if;

if NDC8.CAN_IO_3.DigitalInput3_SteerLimitR_L = TRUE or NDC8.CAN_IO_3.DigitalInput4_SteerLimitR_R = TRUE then
	NDC8.DCD_8.EndLimitSwitchPolarity := 1;
else
	NDC8.DCD_8.EndLimitSwitchPolarity := 0;
end_if;

if NDC8.CAN_IO_3.DigitalInput1_SteerLimitF_L = TRUE or NDC8.CAN_IO_3.DigitalInput2_SteerLimitF_R = TRUE then
	NDC8.DCD_6.EndLimitSwitchPolarity := 1;
else
	NDC8.DCD_6.EndLimitSwitchPolarity := 0;
end_if;

Input.CreepOn := abs(NDC8.VehicleControl.SetSpeed) = NDC8.Vehicle.CreepSpeed;

if  (NDC8.DCD_6.SetAngle > 500 and NDC8.DCD_6.SetAngle <= 8500 and NDC8.DCD_8.SetAngle > 500 and NDC8.DCD_8.SetAngle <= 8500) or
	(NDC8.DCD_6.SetAngle < -500 and NDC8.DCD_6.SetAngle >= -8500 and NDC8.DCD_8.SetAngle < -500 and NDC8.DCD_8.SetAngle >= -8500) then
	Input.SteerMode := 1;
elsif abs(NDC8.DCD_6.SetAngle) > 8500 and abs(NDC8.DCD_6.SetAngle) < 9500
	and abs(NDC8.DCD_8.SetAngle) > 8500 and abs(NDC8.DCD_8.SetAngle) < 9500 then
	Input.SteerMode := 2;
else
	Input.SteerMode := 0;
end_if;

Input.SD_Right := ((NDC8.SegmentTrigger.Bit13_TurnRght_A and NDC8.VehicleControl.Moving)
					or (Input.SteerMode = 0 and NDC8.DCD_6.SetAngle <= -500) (* SD Mode and Right, Just Check Front Wheel *)
					or (Input.SteerMode = 1 and NDC8.VehicleControl.SetSpeed > 0 and NDC8.DCD_6.SetAngle < 0) (* 2*SD Parallel Mode and Right, Just Check Front Wheel  *)
					or (Input.SteerMode = 1 and NDC8.VehicleControl.SetSpeed < 0 and NDC8.DCD_6.SetAngle > 0)) (* 2*SD Parallel Mode and Right, Just Check Front Wheel  *)
					and NDC8.VehicleControl.Moving;

Input.SD_Left :=  ((NDC8.SegmentTrigger.Bit12_TurnLeft_A and NDC8.VehicleControl.Moving)
					or (Input.SteerMode = 0 and NDC8.DCD_6.SetAngle >= 500) (* SD Mode and Left, Just Check Front Wheel *)
					or (Input.SteerMode = 1 and NDC8.VehicleControl.SetSpeed > 0 and NDC8.DCD_6.SetAngle > 0) (* 2*SD Parallel Mode and Left, Just Check Front Wheel  *)
					or (Input.SteerMode = 1 and NDC8.VehicleControl.SetSpeed < 0 and NDC8.DCD_6.SetAngle < 0)) (* 2*SD Parallel Mode and Left, Just Check Front Wheel  *)
					and NDC8.VehicleControl.Moving;

Input.DD_Right := ((Input.SteerMode = 2 and NDC8.VehicleControl.SetSpeed < 0 and NDC8.DCD_6.SetAngle < 0) (* Diff Parallel Mode and Right, Just Check Front Wheel  *)
					or (Input.SteerMode = 2 and NDC8.VehicleControl.SetSpeed > 0 and NDC8.DCD_6.SetAngle > 0)); (* Diff Parallel Mode and Right, Just Check Front Wheel  *)

Input.DD_Left :=  ((Input.SteerMode = 2 and NDC8.VehicleControl.SetSpeed < 0 and NDC8.DCD_6.SetAngle > 0) (* Diff Parallel Mode and Right, Just Check Front Wheel  *)
					or (Input.SteerMode = 2 and NDC8.VehicleControl.SetSpeed > 0 and NDC8.DCD_6.SetAngle < 0)); (* Diff Parallel Mode and Right, Just Check Front Wheel  *)

Input.SD_Forward := ((Input.SteerMode = 0 and NDC8.VehicleControl.SetSpeed > 0 and NDC8.VehicleControl.Moving = TRUE)
					or (Input.SteerMode = 1 and NDC8.VehicleControl.SetSpeed > 0 and NDC8.VehicleControl.Moving = TRUE))
					and (Input.SD_Right = FALSE and Input.SD_Left = FALSE and Input.DD_Right = FALSE and Input.DD_Left = FALSE);

Input.SD_Backward := ((Input.SteerMode = 0 and NDC8.VehicleControl.SetSpeed < 0 and NDC8.VehicleControl.Moving = TRUE)
					or (Input.SteerMode = 1 and NDC8.VehicleControl.SetSpeed < 0 and NDC8.VehicleControl.Moving = TRUE))
					and (Input.SD_Right = FALSE and Input.SD_Left = FALSE and Input.DD_Right = FALSE and Input.DD_Left = FALSE);

INPUT.LoadOnBoard := PLC_RX01_Bit_Load_i;

StopEstopButton := NDC8.SDIO.DigitalInput12_EMO;

END_FUNCTION_BLOCK

(* ---- OUTPUTMAP_FB.ST ---- *)
FUNCTION_BLOCK OUTPUTMAP_FB
VAR_EXTERNAL
NDC8:NDC8_T;
Output : Output_T;
g_PowerOffFlag : BOOL;

END_VAR

VAR_INPUT

END_VAR

VAR_OUTPUT

END_VAR

VAR
	LampBlink : BLINK;

	(* Power Off *)
	PowerOffEvTm : TON;

	BuzzerSyncTm : TON;

	BUZZERMEANS : INT;

END_VAR
(*
------------------------------------------------------------------------------------
 Output_Map_FB
 -----------

 Description:
 Used to map actual outputs to generic variables.

-------------------------------------------------------------------------------------*)

(* In the vehicle documentation, and the OUTPUTS.TYP, more examples of OutputMap_FB is found. * )

NDC8..	:=	OUTPUT.PositionKnownLamp;	( * Green	* )
NDC8..	:=	OUTPUT.EmergencyStopLamp;	( * Red 	* )
NDC8..	:=	OUTPUT.InSystemLamp;		( * Blue	* )
NDC8..	:=	OUTPUT.ResetButtonLamp		( * White	* )
NDC8..	:=	OUTPUT.LoadOnBoardLamp;
NDC8..	:=	OUTPUT.FrontLeftLamp;
NDC8..	:=	OUTPUT.FrontRightLamp;
NDC8..	:=	OUTPUT.RearLeftLamp;
NDC8..	:=	OUTPUT.RearRightLamp;

NDC8..	:=  OUTPUT.ChargPlatesRelay;
NDC8..	:=	OUTPUT.Buzzer;

NDC8..	:=	OUTPUT.ForkRaise;
NDC8..	:=	OUTPUT.ForkLower;

NDC8..	:=	OUTPUT.SafetyScannerAreaControlA1;
NDC8..	:=	OUTPUT.SafetyScannerAreaControlB1;
NDC8..	:=	OUTPUT.SafetyScannerAreaControlA2;
NDC8..	:=	OUTPUT.SafetyScannerAreaControlB2;

OUTPUT.SetValueTraction := NDC8.xCD_x.SetSpeed;      ( * Check FrontWheel.SetSpeedRef and enter it here * )
OUTPUT.SetValueSteer 	:= NDC8.xCD_x.SetAngle;      ( * Check FrontWheel.SetAngleRef and enter it here * )

NDC8.OPT100.Buzzer	:=	OUTPUT.OPTBuzzer;
*)

LampBlink(RUN:= TRUE,  CYCLE:= t#1s);

NDC8.SDIO.DigitalOutput6_LED_INPOS := NDC8.LayoutPosition.InSystem;

NDC8.SDIO.DigitalOutput2_LEDF_L	:=	OUTPUT.FrontLeftLamp;
NDC8.SDIO.DigitalOutput3_LEDF_R	:=	OUTPUT.FrontRightLamp;
NDC8.SDIO.DigitalOutput4_LEDR_L	:=	OUTPUT.RearLeftLamp;
NDC8.SDIO.DigitalOutput5_LEDR_R	:=	OUTPUT.RearRightLamp;

if INPUT.StartMode = TRUE then
	NDC8.SDIO.DigitalOutput7_LED_STR := FALSE;
elsif INPUT.StartMode = FALSE and (INPUT.Manual or g_ErrorCode <> 0) then
	NDC8.SDIO.DigitalOutput7_LED_STR := FALSE;
else
	NDC8.SDIO.DigitalOutput7_LED_STR := LampBlink.Q1;
end_if;

if NDC8.SDIO.DigitalInput5_BTN_BRK = TRUE then
	NDC8.SDIO.DigitalOutput14_LED_BRK := TRUE;
else
	NDC8.SDIO.DigitalOutput14_LED_BRK := FALSE;
end_if;

if g_ErrorCode <> 0 or PLC_RX_Word20_PLC_ErrD <> 0 then
	NDC8.SDIO.DigitalOutput8_LED_RST := LampBlink.Q1;
else
	NDC8.SDIO.DigitalOutput8_LED_RST := FALSE;
end_if;

PowerOffEvTm(IN:= g_PowerOffFlag, PT:= t#600s);

if PowerOffEvTm.Q then
	NDC8.SDIO.DigitalOutput13_PWR_OFF := TRUE;
else
	NDC8.SDIO.DigitalOutput13_PWR_OFF := FALSE;
end_if;

BuzzerSyncTm(IN:=TRUE, PT:=t#10s);

if g_FindSyncFlag = TRUE THEN
	if BuzzerSyncTm.Q = TRUE then
		NDC8.CAN_IO_3.DigitalOutput1_BuzzerCh1 := FALSE;
		NDC8.CAN_IO_3.DigitalOutput2_BuzzerCh2 := FALSE;
		NDC8.CAN_IO_3.DigitalOutput3_BuzzerCh3 := FALSE;
		NDC8.CAN_IO_3.DigitalOutput4_BuzzerCh4 := FALSE;
		BuzzerSyncTm(IN:= FALSE);
	elsif Input.BuzzerByPass = TRUE then
	 	NDC8.CAN_IO_3.DigitalOutput1_BuzzerCh1 := FALSE;
		NDC8.CAN_IO_3.DigitalOutput2_BuzzerCh2 := FALSE;
		NDC8.CAN_IO_3.DigitalOutput3_BuzzerCh3 := FALSE;
		NDC8.CAN_IO_3.DigitalOutput4_BuzzerCh4 := FALSE;
	elsif g_PowerOffFlag = TRUE then (*Ch15*)
		NDC8.CAN_IO_3.DigitalOutput1_BuzzerCh1 := TRUE;
		NDC8.CAN_IO_3.DigitalOutput2_BuzzerCh2 := TRUE;
		NDC8.CAN_IO_3.DigitalOutput3_BuzzerCh3 := TRUE;
		NDC8.CAN_IO_3.DigitalOutput4_BuzzerCh4 := TRUE;
		BUZZERMEANS := 15;
	elsif NDC8.PLC_Application.TxStatusBit9_EStop = TRUE then (*Ch12*)
		NDC8.CAN_IO_3.DigitalOutput1_BuzzerCh1 := FALSE;
		NDC8.CAN_IO_3.DigitalOutput2_BuzzerCh2 := FALSE;
		NDC8.CAN_IO_3.DigitalOutput3_BuzzerCh3 := TRUE;
		NDC8.CAN_IO_3.DigitalOutput4_BuzzerCh4 := TRUE;
		BUZZERMEANS := 12;
	elsif g_ErrorCode <> 0 then (*Ch11*)
		NDC8.CAN_IO_3.DigitalOutput1_BuzzerCh1 := TRUE;
		NDC8.CAN_IO_3.DigitalOutput2_BuzzerCh2 := TRUE;
		NDC8.CAN_IO_3.DigitalOutput3_BuzzerCh3 := FALSE;
		NDC8.CAN_IO_3.DigitalOutput4_BuzzerCh4 := TRUE;
		BUZZERMEANS := 11;
	elsif NDC8.PLC_Application.TxStatusBit12_LostP = TRUE then (*Ch13*)
		NDC8.CAN_IO_3.DigitalOutput1_BuzzerCh1 := TRUE;
		NDC8.CAN_IO_3.DigitalOutput2_BuzzerCh2 := FALSE;
		NDC8.CAN_IO_3.DigitalOutput3_BuzzerCh3 := TRUE;
		NDC8.CAN_IO_3.DigitalOutput4_BuzzerCh4 := TRUE;
		BUZZERMEANS := 13;
	elsif 	NDC8.PLC_Application.TxStatusBit4_LowBatt = TRUE and
		NDC8.SDIO.DigitalOutput12_LEFTMGS = FALSE and
		NDC8.SDIO.DigitalOutput16_RIGHTMGS = FALSE and
		NDC8.PointTrigger.Bit9_Chrg_Right = FALSE and
		NDC8.PointTrigger.Bit10_Chrg_Left = FALSE and
		NDC8.PointTrigger.Bit14_Full_Chrg = FALSE  then (*Ch14*)

		NDC8.CAN_IO_3.DigitalOutput1_BuzzerCh1 := FALSE;
		NDC8.CAN_IO_3.DigitalOutput2_BuzzerCh2 := TRUE;
		NDC8.CAN_IO_3.DigitalOutput3_BuzzerCh3 := TRUE;
		NDC8.CAN_IO_3.DigitalOutput4_BuzzerCh4 := TRUE;
		BUZZERMEANS := 14;
	elsif NDC8.SDIO.DigitalInput3_BMP_O1 = TRUE or NDC8.SDIO.DigitalInput4_BMP_O2 then (*Ch10*)
		NDC8.CAN_IO_3.DigitalOutput1_BuzzerCh1 := FALSE;
		NDC8.CAN_IO_3.DigitalOutput2_BuzzerCh2 := TRUE;
		NDC8.CAN_IO_3.DigitalOutput3_BuzzerCh3 := FALSE;
		NDC8.CAN_IO_3.DigitalOutput4_BuzzerCh4 := TRUE;
		BUZZERMEANS := 10;
	elsif NDC8.PLC_Application.TxStatusBit11_IrStop = TRUE then (*Ch9*)
		NDC8.CAN_IO_3.DigitalOutput1_BuzzerCh1 := TRUE;
		NDC8.CAN_IO_3.DigitalOutput2_BuzzerCh2 := FALSE;
		NDC8.CAN_IO_3.DigitalOutput3_BuzzerCh3 := FALSE;
		NDC8.CAN_IO_3.DigitalOutput4_BuzzerCh4 := TRUE;
		BUZZERMEANS := 9;
	elsif NDC8.PLC_Application.TxStatusBit10_Blocked = TRUE then (*Ch8*)
		NDC8.CAN_IO_3.DigitalOutput1_BuzzerCh1 := FALSE;
		NDC8.CAN_IO_3.DigitalOutput2_BuzzerCh2 := FALSE;
		NDC8.CAN_IO_3.DigitalOutput3_BuzzerCh3 := FALSE;
		NDC8.CAN_IO_3.DigitalOutput4_BuzzerCh4 := TRUE;
		BUZZERMEANS := 8;
	elsif PLC_TX_Word2 <> 0 then (*Ch7*)
		NDC8.CAN_IO_3.DigitalOutput1_BuzzerCh1 := TRUE;
		NDC8.CAN_IO_3.DigitalOutput2_BuzzerCh2 := TRUE;
		NDC8.CAN_IO_3.DigitalOutput3_BuzzerCh3 := TRUE;
		NDC8.CAN_IO_3.DigitalOutput4_BuzzerCh4 := FALSE;
	elsif Input.SafetyScannerSlowDown = TRUE then (*Ch5*)
		NDC8.CAN_IO_3.DigitalOutput1_BuzzerCh1 := TRUE;
		NDC8.CAN_IO_3.DigitalOutput2_BuzzerCh2 := FALSE;
		NDC8.CAN_IO_3.DigitalOutput3_BuzzerCh3 := TRUE;
		NDC8.CAN_IO_3.DigitalOutput4_BuzzerCh4 := FALSE;
		BUZZERMEANS := 5;
	elsif Input.SD_Right or Input.DD_Right then (*Ch4*)
		NDC8.CAN_IO_3.DigitalOutput1_BuzzerCh1 := FALSE;
		NDC8.CAN_IO_3.DigitalOutput2_BuzzerCh2 := FALSE;
		NDC8.CAN_IO_3.DigitalOutput3_BuzzerCh3 := TRUE;
		NDC8.CAN_IO_3.DigitalOutput4_BuzzerCh4 := FALSE;
	elsif Input.SD_Left or Input.DD_Left then (*Ch3*)
		NDC8.CAN_IO_3.DigitalOutput1_BuzzerCh1 := TRUE;
		NDC8.CAN_IO_3.DigitalOutput2_BuzzerCh2 := TRUE;
		NDC8.CAN_IO_3.DigitalOutput3_BuzzerCh3 := FALSE;
		NDC8.CAN_IO_3.DigitalOutput4_BuzzerCh4 := FALSE;
	elsif Input.SD_Backward then (*Ch2*)
		NDC8.CAN_IO_3.DigitalOutput1_BuzzerCh1 := FALSE;
		NDC8.CAN_IO_3.DigitalOutput2_BuzzerCh2 := TRUE;
		NDC8.CAN_IO_3.DigitalOutput3_BuzzerCh3 := FALSE;
		NDC8.CAN_IO_3.DigitalOutput4_BuzzerCh4 := FALSE;
		BUZZERMEANS := 2;
	elsif Input.SD_Forward then (*Ch1*)
		NDC8.CAN_IO_3.DigitalOutput1_BuzzerCh1 := TRUE;
		NDC8.CAN_IO_3.DigitalOutput2_BuzzerCh2 := FALSE;
		NDC8.CAN_IO_3.DigitalOutput3_BuzzerCh3 := FALSE;
		NDC8.CAN_IO_3.DigitalOutput4_BuzzerCh4 := FALSE;
	elsif NDC8.Automatic.ExecDriveCommand = TRUE then (*Ch1*)
		NDC8.CAN_IO_3.DigitalOutput1_BuzzerCh1 := TRUE;
		NDC8.CAN_IO_3.DigitalOutput2_BuzzerCh2 := FALSE;
		NDC8.CAN_IO_3.DigitalOutput3_BuzzerCh3 := FALSE;
		NDC8.CAN_IO_3.DigitalOutput4_BuzzerCh4 := FALSE;
		BUZZERMEANS := 1;

	(*Ch6*)
	(*
	elsif (StopWord <> 0 and not StopStartDelay and not StopCharge and not StopLoadOP) or (StopWord2 <> 0 and not StopByBCD and not StopRobotNotIdle )then
		NDC8.CAN_IO_3.DigitalOutput1_BuzzerCh1 := FALSE;
		NDC8.CAN_IO_3.DigitalOutput2_BuzzerCh2 := TRUE;
		NDC8.CAN_IO_3.DigitalOutput3_BuzzerCh3 := TRUE;
		NDC8.CAN_IO_3.DigitalOutput4_BuzzerCh4 := FALSE;*)

	else
		NDC8.CAN_IO_3.DigitalOutput1_BuzzerCh1 := FALSE;
		NDC8.CAN_IO_3.DigitalOutput2_BuzzerCh2 := FALSE;
		NDC8.CAN_IO_3.DigitalOutput3_BuzzerCh3 := FALSE;
		NDC8.CAN_IO_3.DigitalOutput4_BuzzerCh4 := FALSE;
		BUZZERMEANS := 0;
	end_if;
end_if;

END_FUNCTION_BLOCK

(* ---- MAIN.ST ---- *)
PROGRAM MAIN
VAR_EXTERNAL
	NDC8:NDC8_T;

(* Function blocks available from all programs. *)
	DisplayStopString : DisplayStopString_FB;
	EventQueue : EventQueue_FB;

END_VAR

VAR
(* Standard functions *)
	Indicators : Indicators_FB;
	Mode : ModeControl_FB ;
	Navigation : Navigation_FB;
	StopWordFB : StopWord_FB;
	TX_Status : TX_Status_FB;
	EventHandler : EVENTHANDLER_FB;
	AutoLoad : AutoLoad_FB;
	CarrierControl:CarrierControl_FB;
	Display : Display_FB;
	OPTX2  : OPTX2_FB;
	LS2000 : LS2000_FB;
	DebugFB : Debug_FB;
	NavInit : NavInit_FB;
	PLC_Communication : PLC_Communication_FB;

	F_SteerSupervision : DRIVERSUPERVISION_FB;
	F_DriveSupervision : DRIVERSUPERVISION_FB;
	R_SteerSupervision : DRIVERSUPERVISION_FB;
	R_DriveSupervision : DRIVERSUPERVISION_FB;
	BMS_CHG : BMS_CHG_FB;

	VehicleMovingFlag : BOOL;

(* Error Trigger BlackBox *)
	Error_Set_Trig : BOOL;
	Error_BB_TrigR : R_Trig;
	Error_Trig : BOOL;

(* OM-PLC Trigger BlackBox *)
	OMPLC_BB_TrigR : R_Trig;
	OMPLC_Trig : BOOL;

	BlackBox : BlackBox_FB;
(* Master Link *)
	MasterLinkR : R_Trig;

(* Vehicle specific functions *)
	InputMap : InputMap_fb;
	OutputMap : OutputMap_fb;

(* PLC Communication Check *)
	LastCommCheckFlag : BOOL;

	CommCheckTimeUp : TON;

	iVar1 : INT;

(* Blocking Power Off Check *)
	BlockPowOffTm : TON;
	BlockPowOffTmValue : TIME;

(* Lost Power Off Check *)
	LostPosPowOffTm : TON;
	LostPosPowOffTmValue : TIME;

(* Over Voltage ESTOP *)

(* Error Power Off Check *)
	ErrorOccurFlag : BOOL;
	ErrorPowOffTm : TON;
	ErrorPowOffTmValue : TIME;

(* Battery Low OT *)
	BatLowTm : TON;

(* Display Error String *)
	FailCodeDint : dint;

	BbxTrig_FT : F_trig;
	ExecDriveCommand_RT : R_Trig;
	FailTimerTON : TON;

	PreviousMainState,
	PreviousLoadState,
	PreviousUnLoadState,
	PreviousTravelDir,
	PreviousFailCode,
	PreviousForkHeight,

	PreviousExecDriveCommand,
	PreviousCancelOperation,
	bbxtrigger			:bool;

(* All OK Motor Find Z-phase *)
	AllOK_R :R_Trig;
	AllOK_Delay : TON;

	FindSyncDelay : TON;

	FindSyncStep : INT := 0;

	CurPnt : DINT := 0;
	CurSeg : DINT := 0;

(* Navigation Down Timer Check *)
	NavLevelDown_Start : BOOL;
	NavLevelDown_TM : TON;
	NavLevelDown_TmUp	 : BOOL;

(* LS2000 Attached Timer *)
	LS2000_Attached_M : TON;

(* AGV Travel Distance Sampling Timer *)
	LastEncoderDistance : UINT := 0;
	CurrentEncoderDistance : UINT := 0;
	TravelDistanceSamplingTimer : TON;

(* Black Box Trigger *)
	BootUpDelay : TON;
	NoErrorDelay : TON;

	ErrorFlag : bool;
	ErrorTrigFlag : bool;
	ErrorTrigR : R_Trig;

	ErrorCodeString : string;
	BBMessage : string;

(* Update Data *)
	DataUpdate : DataUpload_FB;
(* Check Steering Sync State  *)
	SteerEncoderNormalStatus : BOOL;
	Z_PHASE_REALLY_NG_T : TON;
	MovingDoneLT : F_Trig;
	ChanceToSyncFailCount : DINT := 0;
(* Position Lost Delay , InSystem too slow *)
	PosLostTimer : TON;
	IsInSystemFlag : BOOL := FALSE;
END_VAR
(*

MAIN
--------

These function blocks are a minimum to run a typical Steer/drive fork truck.

*)

AllOK_R(CLK:=NDC8.SDIO.AllOK_DigitalOutput1);

if AllOK_R.Q and NDC8.SDIO.DigitalInput2_BTN_RST = FALSE then
	g_StartFindSync:= TRUE;
	StopFindSync := TRUE;
elsif AllOK_R.Q and NDC8.SDIO.DigitalInput2_BTN_RST = TRUE then
	g_StartFindSync := FALSE;
	g_FindSyncFlag := TRUE;
	StopFindSync := FALSE;
end_if;

if NDC8.CAN_IO_3.DigitalInput5_LIMF_O = TRUE then
	NDC8.DCD_6.SyncGate := TRUE;
else
	NDC8.DCD_6.SyncGate := FALSE;
end_if;

if NDC8.CAN_IO_3.DigitalInput6_LIMR_O = TRUE then
	NDC8.DCD_8.SyncGate := TRUE;
else
	NDC8.DCD_8.SyncGate := FALSE;
end_if;

AllOK_Delay(IN:=g_StartFindSync, PT:=t#5s);

if AllOK_Delay.Q and g_FindSyncFlag = FALSE and NDC8.SDIO.DigitalInput2_BTN_RST = FALSE then
	case FindSyncStep of
	0:
	(* Steer Turn to 2000 *)
	NDC8.Manual.PlcSelect := true;
	NDC8.Manual.PLCAngle := -9000;
	NDC8.Manual.PlcSetOperationMode := 1;
	NDC8.Manual.PLCSteerMode := 0;
	NDC8.Manual.PlcSelectMask 		:= 2#10101;
	INPUT.Manual := TRUE;
	PLC_RX_Word16_BMS_BatV := 540;(*Prevent Cold Start LowBat*)

	FindSyncDelay(IN:=TRUE, PT:=t#5s);
	if FindSyncDelay.Q then
		FindSyncStep := 1;
		FindSyncDelay(IN:=FALSE);
	end_if;

	1:
	(* Steer Turn to -2000 *)
	NDC8.Manual.PlcSelect := true;
	NDC8.Manual.PLCAngle := 9000;
	NDC8.Manual.PlcSetOperationMode := 1;
	NDC8.Manual.PLCSteerMode := 0;
	NDC8.Manual.PlcSelectMask 		:= 2#10101;

	FindSyncDelay(IN:=TRUE, PT:=t#5s);
	if FindSyncDelay.Q then
		FindSyncStep := 2;
		FindSyncDelay(IN:=FALSE);
	end_if;

	2:
	(* Steer Turn to 0 *)
	NDC8.Manual.PlcSelect := true;
	NDC8.Manual.PLCAngle := 0;
	NDC8.Manual.PlcSetOperationMode := 0;
	NDC8.Manual.PLCSteerMode := 0;
	NDC8.Manual.PlcSelectMask 		:= 2#10101;

	FindSyncDelay(IN:=TRUE, PT:=t#7s);
	if FindSyncDelay.Q then
		FindSyncStep := 3;
		FindSyncDelay(IN:=FALSE);
		IF NDC8.DCD_6.EncoderStatus = 1 AND NDC8.DCD_8.EncoderStatus = 1 THEN
			g_FindSyncFlag := TRUE;
			NDC8.Manual.PlcSelectMask := 0;
			g_StartFindSync := FALSE;
			StopFindSync := FALSE;
		END_IF;
	end_if;
	3:
	(* Check Encoder Status *)
	IF NDC8.DCD_6.EncoderStatus = 0 OR NDC8.DCD_8.EncoderStatus = 0 THEN
		FindSyncStep := 0;
	ELSE
	 	FindSyncStep := 4;
	END_IF;
	end_case;

end_if;

IF INPUT.Reset_PB THEN
	StopStartDelay := 0;
END_IF;

(* Check Steering Sync State  *)

SteerEncoderNormalStatus := NDC8.DCD_6.EncoderStatus = 1 AND NDC8.DCD_8.EncoderStatus = 1;

IF NDC8.UserDefined.Integer32_10_ChanceToSyncFailLimit = 0 THEN
	NDC8.UserDefined.Integer32_10_ChanceToSyncFailLimit := 10;
END_IF;

MovingDoneLT(CLK := NDC8.Automatic.ExecDriveCommand);

IF MovingDoneLT.Q = TRUE AND SteerEncoderNormalStatus = FALSE THEN
	ChanceToSyncFailCount := ChanceToSyncFailCount + 1;
END_IF;

IF MovingDoneLT.Q = TRUE AND SteerEncoderNormalStatus = TRUE THEN
	ChanceToSyncFailCount := 0;
END_IF;

if NDC8.CanOpenMaster.NMTState = 5 and NDC8.CanOpenMaster.State = 0 then

(* INPUTS *)
	InputMap();					(* Mapping inputs on devices to generic names *)

(*Decisionmaking PLC:s*)

	Autoload();	 (* Load handling 		*)

	LS2000();

	CarrierControl(	LS2000Slowdown := LS2000.Slowdown);

	if g_StartFindSync = FALSE then
		Mode();												(* Selects vehicle mode *)
	end_if;

(* OUTPUTS *)
	OutputMap();				(* Mapping outputs on devices to generic names *)

(* BMS Charger *)
	BMS_CHG();

	PLC_Communication();
end_if;

(* These FB can be run also during startup and in safe state *)

	(* Information *)
Timer();						(* Square wave timers 										*)

Navigation(AutoInsertNotInsideTargetSafety := CarrierControl.AutoInsertNotInsideTargetSafety);					(* Info regarding navigation 								*)

StopWordFB();					(* Stop reasons 											*)

DisplayStopString();			(* Displays user defined stop reasons on the display 		*)

TX_Status();					(* Sends status bits to Master Controller 					*)

EventHandler();					(* Transmits events from the queue							*)

debugFB();

Indicators(	AutoInsertNotInsideTargetSafety := CarrierControl.AutoInsertNotInsideTargetSafety,
			AutoinsertInProgress 	:= CarrierControl.AutoinsertInProgress,
			StartDelayStartWarning 	:= CarrierControl.StartDelayStartWarning,
			LS2000SlowDown 			:= false);						(* Controls lamps and buzzers 								*)

(*System Brake Signal*)
if NDC8.UserDefined.Braker_Signal = FALSE or (INPUT.Manual = TRUE and NDC8.SDIO.DigitalInput5_BTN_BRK = TRUE) or (INPUT.Auto = TRUE and NDC8.SDIO.DigitalInput5_BTN_BRK = TRUE) then
	(*Brake Release*)
	NDC8.DCD_5.DigitalOutput2_Braker := TRUE;
	NDC8.DCD_7.DigitalOutput2_Braker := TRUE;
else
	(*Brake Lock*)
	NDC8.DCD_5.DigitalOutput2_Braker := FALSE;
	NDC8.DCD_7.DigitalOutput2_Braker := FALSE;
end_if;

if INPUT.Auto = TRUE and NDC8.SDIO.DigitalInput5_BTN_BRK = TRUE and NDC8.Mcd.Button8 = FALSE then
	StopAutoBrakeRelease := TRUE;
else
	StopAutoBrakeRelease := FALSE;
end_if;

(* Encoder Supervision *)
VehicleMovingFlag := NDC8.VehicleControl.Moving and not NDC8.PLC_Application.TxStatusBit9_EStop and StopWord = 0 and StopWord2 = 0;

F_SteerSupervision(Command:= NDC8.DCD_6.SetAngle,FeedBack:= NDC8.DCD_6.WheelAngle,Range:= 1000,Timeout:= t#30s,Moving:= VehicleMovingFlag);
R_SteerSupervision(Command:= NDC8.DCD_8.SetAngle,FeedBack:= NDC8.DCD_8.WheelAngle,Range:= 1000,Timeout:= t#30s,Moving:= VehicleMovingFlag);

F_DriveSupervision(Command:= NDC8.DCD_5.SetSpeed,FeedBack:= NDC8.DCD_5.DriveEncSpeed,Range:= 100,Timeout:= t#30s,Moving:= VehicleMovingFlag);
R_DriveSupervision(Command:= NDC8.DCD_7.SetSpeed,FeedBack:= NDC8.DCD_7.DriveEncSpeed,Range:= 100,Timeout:= t#30s,Moving:= VehicleMovingFlag);

(* OM-PLC Bit*)

	(*OM_PLC_W1_Bit_WaitCharge		:= FALSE;*)
	(*OM_PLC_W1_Bit_WaitOrder			:= FALSE;*)

	OM_PLC_Word1 := INT_TO_WORD(NDC8.OMPLC.ChargeOM);
	OM_PLC_Word2 := INT_TO_WORD(NDC8.OMPLC.Stop_OM);

	StopByOM_PLC := OM_PLC_W2_Bit_SetEmgStop;

	(*OM_PLC_W2_Bit_BCD_setReq		:= FALSE;*)
	(*OM_PLC_W2_Bit_BCD_setOK			:= FALSE;*)
	(*OM_PLC_W2_Bit_BCD_Init			:= FALSE;*)
	(*OM_PLC_W2_Bit_BCD_NoRead		:= FALSE;*)
	(*OM_PLC_W2_Bit_Set_Result		:= FALSE;*)
	(*OM_PLC_W2_Bit_Err_Comp			:= FALSE;*)
	(*OM_PLC_W2_Bit_Err_BCR			:= FALSE;*)
	(*OM_PLC_W2_Bit_SetT10Terr		:= FALSE;*)

	g_PowerOffFlag_OMPLC := OM_PLC_W2_Bit_PowerOffOm;

	(*OM_PLC_W2_Bit_SetCondErr		:= FALSE;*)
	(*OM_PLC_W2_Bit_SetT30TErr		:= FALSE;*)

	OMPLC_BB_TrigR(CLK:= OM_PLC_W2_Bit_BB_setReq);

	if OMPLC_BB_TrigR.Q = TRUE then
		OMPLC_Trig := TRUE;
	end_if;

	if OMPLC_Trig = TRUE then
		NDC8.BlackBox.TrigReason:= 'OM_PLC';
		BlackBox();
		if BlackBox.Finished then
			OMPLC_Trig := FALSE;
		end_if;
	end_if;

	(*OM_PLC_W2_Bit_Set_LowTS			:= FALSE;*)
	(*OM_PLC_W2_Bit_SetHOErr			:= FALSE;*)

	OM_PLC_W7_Bit_Area1 := NDC8.SegmentTrigger.Bit4_Area1_Seg;
	OM_PLC_W7_Bit_Area2 := NDC8.SegmentTrigger.Bit5_Area2_Seg;
	OM_PLC_W7_Bit_Area4 := NDC8.SegmentTrigger.Bit6_Area4_Seg;
	OM_PLC_W7_Bit_Area8 := NDC8.SegmentTrigger.Bit7_Area8_Seg;

	(* OM-PLC Word*)
	NDC8.OMPLC.ChargeOM := WORD_TO_INT(OM_PLC_Word1);
	NDC8.OMPLC.Stop_OM := WORD_TO_INT(OM_PLC_Word2);

	if NDC8.LayoutPosition.Point <> 0 then
		CurPnt := NDC8.LayoutPosition.Point;
	end_if;

	if NDC8.LayoutPosition.Segment <> 0 then
		CurSeg := NDC8.LayoutPosition.Segment;
	end_if;

	NDC8.OMPLC.Cur_Pnt := DINT_TO_INT(CurPnt);
	NDC8.OMPLC.Cur_Seg := DINT_TO_INT(CurSeg);

	OM_PLC_Word7 := INT_TO_WORD(NDC8.OMPLC.Drv_Area);

	OM_PLC_W7_Bit_Area1 := NDC8.SegmentTrigger.Bit4_Area1_Seg;
	OM_PLC_W7_Bit_Area2 := NDC8.SegmentTrigger.Bit5_Area2_Seg;
	OM_PLC_W7_Bit_Area4 := NDC8.SegmentTrigger.Bit6_Area4_Seg;
	OM_PLC_W7_Bit_Area8 := NDC8.SegmentTrigger.Bit7_Area8_Seg;

	NDC8.OMPLC.Drv_Area := WORD_TO_INT(OM_PLC_Word7);

(* Alarm code *)

if LastCommCheckFlag = PLC_RX01_Bit_ChkCom_RX then
	CommCheckTimeUp(IN:= TRUE, PT:= t#10s);
	if CommCheckTimeUp.Q then
		g_PlcComLinkUp := FALSE;
	end_if;
else
	LastCommCheckFlag := PLC_RX01_Bit_ChkCom_RX;
	CommCheckTimeUp(IN:= FALSE);
	g_PlcComLinkUp := TRUE;
end_if;

if g_FindSyncFlag = TRUE then

OM_PLC_Word1 := INT_TO_WORD(NDC8.OMPLC.ChargeOM);
OM_PLC_Word2 := INT_TO_WORD(NDC8.OMPLC.Stop_OM);

	MasterLinkR(CLK:= NDC8.Master.MasterLinkUp);

	if MasterLinkR.Q or g_AGV_ErrorReset or (NDC8.Mcd.Button8 = TRUE and INPUT.Manual = TRUE) THEN (* When Master Link up, Error Status need to be update again *)
		g_ErrorCode := 0;
		PLC_TX_Word13_STr_Err := 0;
		OM_PLC_W2_Bit_SetEmgStop := FALSE;
		FORCECOUNT := FORCECOUNT + 1;
	elsif PLC_RX_Word20_PLC_ErrD <> 0 and g_ErrorCode = 0 then
		g_ErrorCode := PLC_RX_Word20_PLC_ErrD;
	elsif PLC_RX14_Bit_BMS_Short then
		g_ErrorCode := 101;
	elsif PLC_RX14_Bit_BMS_Over then
		g_ErrorCode := 102;
(*	elsif PLC_RX03_Bit_STwDisBMS1 <> 0 or PLC_RX03_Bit_STwDisBMS2 <> 0 then  G5 CHARGE OVER VOLTAGE ,HOWEVER WITH BMS ACTIVE ITS NO USE
		if PLC_RX_Word16_BMS_BatV > 700 then
			g_ErrorCode := 102;
		end_if;*)
	elsif PLC_RX14_Bit_BMS_TempEr then
		g_ErrorCode := 103;
	elsif PLC_RX14_Bit_BMS_LowV then
		g_ErrorCode := 104;
	elsif PLC_RX14_Bit_BMS_Ch_Err and PLC_RX03_Bit_STw_EnaChg then
		g_ErrorCode := 105;
	elsif PLC_RX14_Bit_BMS_Thermi then
		g_ErrorCode := 106;
	elsif PLC_RX14_Bit_BMS_CT then
		g_ErrorCode := 107;
	elsif PLC_RX14_Bit_BMS_Couple then
		g_ErrorCode := 108;
	elsif PLC_RX14_Bit_BMS_Bat then
		g_ErrorCode := 109;
	elsif PLC_RX14_Bit_BMS_NG then
		g_ErrorCode := 110;
	elsif F_DriveSupervision.NotMovingFail = TRUE then
		g_ErrorCode := 122;
	elsif R_DriveSupervision.NotMovingFail = TRUE then
		g_ErrorCode := 123;
	elsif (F_SteerSupervision.NotMovingFail = TRUE or R_SteerSupervision.NotMovingFail = TRUE) AND g_StartFindSync or (NDC8.DCD_6.EncoderStatus = 0 or NDC8.DCD_8.EncoderStatus = 0) AND g_StartFindSync THEN
		g_ErrorCode := 124;
	elsif ChanceToSyncFailCount > NDC8.UserDefined.Integer32_10_ChanceToSyncFailLimit THEN
		g_ErrorCode := 124;
	elsif g_BattLim_NG then
		g_ErrorCode := 127;
	(*elsif not NDC8.DCD_5.DigitalInput2_OverRelayFS or not NDC8.DCD_5.DigitalInput3_OverRelayFD or not NDC8.DCD_7.DigitalInput2_OverRelayRS or not NDC8.DCD_7.DigitalInput3_OverRelayRD then*)
	elsif not NDC8.DCD_5.DigitalInput3_OverRelayFD or not NDC8.DCD_7.DigitalInput3_OverRelayRD then
		g_ErrorCode := 131;
	elsif NDC8.SDIO.DigitalInput3_BMP_O1 = TRUE or NDC8.SDIO.DigitalInput4_BMP_O2 = TRUE or NDC8.SDIO.DigitalInput8_BMP_E = FALSE then
		g_ErrorCode := 132;
	elsif NDC8.SDIO.DigitalInput12_EMO = FALSE then
		g_ErrorCode := 133;
	elsif NDC8.Autoinsert.StatusID = 5 then
		g_ErrorCode := 136;
	elsif NDC8.LayoutPosition.InSystem = FALSE AND STARTENABLE AND (PLC_TX01_Bit_HostMode = TRUE or PLC_TX01_Bit_LocalMode = TRUE) AND CarrierControl.AutoinsertInProgress = false THEN
		IsInSystemFlag := NOT NDC8.Mcd.Button1;
		PosLostTimer(IN := IsInSystemFlag, PT := t#2s);
		IF PosLostTimer.Q THEN
			g_ErrorCode := 137;
			PosLostTimer(IN := FALSE);
		END_IF;
	elsif NDC8.Guidance.OutsideSafetyZone = TRUE then
		g_ErrorCode := 138;
	elsif NDC8.LS2000.Connected = FALSE or NDC8.LS2000.Attached = FALSE or NDC8.LS2000.NavActive = FALSE then
		g_ErrorCode := 139;
	elsif NavLevelDown_TmUp = TRUE then
		g_ErrorCode := 140;
	elsif OM_PLC_W2_Bit_SetEmgStop = TRUE then
		g_ErrorCode := 145;
	elsif not NDC8.CAN_IO_3.DigitalInput1_SteerLimitF_L or not NDC8.CAN_IO_3.DigitalInput2_SteerLimitF_R or not NDC8.CAN_IO_3.DigitalInput3_SteerLimitR_L or not NDC8.CAN_IO_3.DigitalInput4_SteerLimitR_R then
		g_ErrorCode := 161;
	elsif (PLC_RX01_Bit_ChrgEmg and PLC_TX01_Bit_ManMode) or (PLC_RX01_Bit_ChrgEmg and not PLC_TX01_Bit_ManMode and NDC8.PLC_Application.TxStatusBit6_Charge) then
		g_ErrorCode := 174;
	elsif F_DriveSupervision.OverRangeFail = TRUE then
		g_ErrorCode := 182;
	elsif R_DriveSupervision.OverRangeFail = TRUE then
		g_ErrorCode := 183;
	elsif g_ChargeOverTime = TRUE then
		g_ErrorCode := 185;
	elsif NDC8.Automatic.ExecDriveCommand = TRUE and PLC_RX01_Bit_EnableLD_i = FALSE then
		(*g_ErrorCode := 190;*)
		;

	elsif NDC8.CanOpenMaster.State = 1 and NDC8.CanOpenMaster.EMCY_BusID = 1 and NDC8.CanOpenMaster.EMCY_NodeID = 2 then
		g_ErrorCode := 194;
		StopByCanErr_Node2 := TRUE;
	elsif NDC8.CanOpenMaster.State = 1 and NDC8.CanOpenMaster.EMCY_BusID = 1 and NDC8.CanOpenMaster.EMCY_NodeID = 3 then
		g_ErrorCode := 195;
		StopByCanErr_Node3 := TRUE;
	elsif NDC8.CanOpenMaster.State = 1 and NDC8.CanOpenMaster.EMCY_BusID = 1 and NDC8.CanOpenMaster.EMCY_NodeID = 5 then
		g_ErrorCode := 197;
		StopByCanErr_Node5 := TRUE;
	elsif NDC8.CanOpenMaster.State = 1 and NDC8.CanOpenMaster.EMCY_BusID = 1 and NDC8.CanOpenMaster.EMCY_NodeID = 6 then
		g_ErrorCode := 198;
		StopByCanErr_Node6 := TRUE;
	elsif NDC8.CanOpenMaster.State = 1 and NDC8.CanOpenMaster.EMCY_BusID = 1 and NDC8.CanOpenMaster.EMCY_NodeID = 7 then
		g_ErrorCode := 199;
		StopByCanErr_Node7 := TRUE;
	elsif NDC8.CanOpenMaster.State = 1 and NDC8.CanOpenMaster.EMCY_BusID = 1 and NDC8.CanOpenMaster.EMCY_NodeID = 8 then
		g_ErrorCode := 200;
		StopByCanErr_Node8 := TRUE;
	elsif CommCheckTimeUp.Q = TRUE then
		g_ErrorCode := 383;
	elsif Autoload.Fail = TRUE then
		;
		(*When Autoload Fail, ErrorCode Set by AutoLoad_FB, Here do nothing *)
		(*After Report event code in AutoLoad, "Fail" will reset in Step 1000*)
	else
		(*_ErrorCode := 0;*)
		(* only use Reset PB to Clear Error Code *)
		;
	end_if;

	if g_ErrorCode > 100 and g_ErrorCode < 201 then
		PLC_TX_Word13_STr_Err := g_ErrorCode;
	end_if;

	NDC8.OMPLC.ChargeOM := WORD_TO_INT(OM_PLC_Word1);
	NDC8.OMPLC.Stop_OM := WORD_TO_INT(OM_PLC_Word2);

end_if;

(* Error Trigger Black Box *)
if PLC_TX01_Bit_HostMode and (g_ErrorCode = 131 or g_ErrorCode = 132 or g_ErrorCode = 133 or g_ErrorCode = 138 or g_ErrorCode = 137 or g_ErrorCode = 140 or g_ErrorCode = 161) then
	Error_Set_Trig := true;
else
	Error_Set_Trig := false;
end_if;

Error_BB_TrigR(CLK:= Error_Set_Trig);

if Error_BB_TrigR.Q = TRUE then
	Error_Trig := TRUE;
end_if;

if Error_Trig = TRUE then
	ErrorCodeString := WORD_TO_STRING(g_ErrorCode);
	BBMessage := CONCAT('AGV_Error_', ErrorCodeString);
	NDC8.BlackBox.TrigReason := BBMessage;
	BlackBox();
	if BlackBox.Finished then
		Error_Trig := FALSE;
	end_if;
end_if;

if g_ErrorCode <> 0 then
	StopByErrorCode := TRUE;
else
	StopByErrorCode := FALSE;
end_if;

if (PLC_RX01_Bit_EnableLD_i = FALSE or Input.StartMode = FALSE) and Input.Auto then
	StopRobotNotIdle := TRUE;
else
	StopRobotNotIdle := FALSE;
end_if;

(* Blocking Power Off Check *)
BlockPowOffTmValue := DINT_TO_TIME(NDC8.UserDefined.Integer32_52_PowOffTm);
LostPosPowOffTmValue := DINT_TO_TIME(NDC8.UserDefined.Integer32_52_PowOffTm);

BlockPowOffTm(IN := NDC8.PLC_Application.TxStatusBit10_Blocked, PT := BlockPowOffTmValue);
if NDC8.UserDefined.Boolean_10_BlockPowOffEn = TRUE and PLC_TX01_Bit_HostMode = TRUE then
	if BlockPowOffTm.Q = TRUE then
		g_PowerOffFlag_Block := TRUE;
	else
		g_PowerOffFlag_Block := FALSE;
	end_if;
else
	g_PowerOffFlag_Block := FALSE;
end_if;

(* Navigation Level Down Check *)
if NDC8.Position.NavLevel < 45 and INPUT.Auto = TRUE then
	NavLevelDown_Start := TRUE;
else
	NavLevelDown_Start := FALSE;
	NavLevelDown_TmUp := FALSE;
end_if;

NavLevelDown_TM(IN := NavLevelDown_Start, PT := t#60s);

if NavLevelDown_TM.Q = TRUE then
	NavLevelDown_TmUp := TRUE;
end_if;

(* Lost Power Off Check *)
LostPosPowOffTm(IN := NDC8.PLC_Application.TxStatusBit12_LostP, PT := LostPosPowOffTmValue);
if NDC8.UserDefined.Boolean_11_LostPosPowOffEn = TRUE and PLC_TX01_Bit_HostMode = TRUE then
	if LostPosPowOffTm.Q = TRUE then
		g_PowerOffFlag_Lost := TRUE;
	else
		g_PowerOffFlag_Lost := FALSE;
	end_if;
else
	g_PowerOffFlag_Lost := FALSE;
end_if;

(* Error Power Off Check *)
if g_ErrorCode <> 0 then
	ErrorOccurFlag := TRUE;
else
	ErrorOccurFlag := FALSE;
end_if;

ErrorPowOffTm(IN := ErrorOccurFlag, PT := t#600s);
if PLC_TX01_Bit_HostMode = TRUE then
	if ErrorPowOffTm.Q = TRUE then
		g_PowerOffFlag_Error := TRUE;
	else
		g_PowerOffFlag_Error := FALSE;
	end_if;
else
	g_PowerOffFlag_Error := FALSE;
end_if;

(* Battery Low OT *)
if PLC_RX04_Bit_STw_LowOT or g_ErrorCode = 102 then
	StopBatLowOT := TRUE;
	if VehicleMovingFlag = FALSE
		and  NDC8.LoadDocking.OnTarget = FALSE
		and PLC_TX01_Bit_ManMode = FALSE
		and NDC8.SDIO.DigitalOutput16_RIGHTMGS = FALSE
		and NDC8.SDIO.DigitalOutput12_LEFTMGS = FALSE THEN
		g_BattLim_NG := TRUE;
		BatLowTm(IN := TRUE, PT := t#10s);
		if BatLowTm.Q then
			g_PowerOffFlag_PLC := TRUE;
		end_if;
	else
		BatLowTm(IN := FALSE);
		g_PowerOffFlag_PLC := FALSE;
	end_if;
else
	BatLowTm(IN := FALSE);
	g_PowerOffFlag_PLC := FALSE;
	StopBatLowOT := FALSE;
end_if;

g_PowerOffFlag := g_PowerOffFlag_Error or g_PowerOffFlag_Block or g_PowerOffFlag_Lost or g_PowerOffFlag_PLC or g_PowerOffFlag_OMPLC or g_PowerOffFlag_OP;

(* Display Stop String update *)
InStatus 			:= g_ErrorCode<>0;
FailCodeDint		:= WORD_TO_DINT(g_ErrorCode);
DisplayStopString(INStatus:=InStatus, StopString:=49, StopValue:=FailCodeDint);		(* Failcode *)

(* IR Sensor switch always on *)
NDC8.CAN_IO_3.DigitalOutput9_AreaF_SW1 := TRUE;
NDC8.CAN_IO_3.DigitalOutput10_AreaF_SW2 := TRUE;
NDC8.CAN_IO_3.DigitalOutput13_AreaR_SW1 := TRUE;
NDC8.CAN_IO_3.DigitalOutput14_AreaR_SW2 := TRUE;

(* IR Speed Control *)

if NDC8.SegmentTrigger.Bit15_DisIrStop = FALSE and (NDC8.SegmentTrigger.Bit14_DisIrSlow = FALSE and PLC_TX01_Bit_ManMode = FALSE) then

	if ((NDC8.CAN_IO_3.DigitalInput9_AreaF_IN1 = FALSE and NDC8.VehicleControl.TravelDir = 1)
		or (NDC8.CAN_IO_3.DigitalInput13_AreaR_IN1 = FALSE and NDC8.VehicleControl.TravelDir = 0) )
		and NDC8.Automatic.ExecDriveCommand and StopAutoBrakeRelease = FALSE then
		Input.SafetyScannerSlowDown := TRUE;
	else
		Input.SafetyScannerSlowDown := FALSE;
	end_if;

else
	Input.SafetyScannerSlowDown := FALSE;

end_if;

if NDC8.SegmentTrigger.Bit15_DisIrStop = FALSE and PLC_TX01_Bit_ManMode = FALSE then

	if ((NDC8.CAN_IO_3.DigitalInput10_AreaF_IN2 = FALSE and NDC8.VehicleControl.TravelDir = 1)
		or (NDC8.CAN_IO_3.DigitalInput14_AreaR_IN2 = FALSE and NDC8.VehicleControl.TravelDir = 0))
		and NDC8.Automatic.ExecDriveCommand and StopAutoBrakeRelease = FALSE then
		StopObstacle := TRUE;
	else
		StopObstacle := FALSE;
	end_if;

	if StopObstacle = TRUE and NDC8.Mcd.Button7 = TRUE then
		StopObstacle := FALSE;
	end_if;

else
	StopObstacle := FALSE;

end_if;

if NDC8.LS2000.Attached = true then
	LS2000_Attached_M(IN:=TRUE, PT:=t#60s);
else
	LS2000_Attached_M(IN:=FALSE);
end_if;

if LS2000_Attached_M.Q = TRUE then
	LS2000_Attached_M(IN:=FALSE);
	NDC8.UserDefined.Integer32_60_LS2000_Attached_M := NDC8.UserDefined.Integer32_60_LS2000_Attached_M + 1;
end_if;

if NDC8.UserDefined.Integer32_60_LS2000_Attached_M > 60 then
	NDC8.UserDefined.Integer32_59_LS2000_Attached_H := NDC8.UserDefined.Integer32_59_LS2000_Attached_H + 1;
	NDC8.UserDefined.Integer32_60_LS2000_Attached_M := 0;
end_if;

if NDC8.UserDefined.Integer32_59_LS2000_Attached_H > 24 then
	NDC8.UserDefined.Integer32_58_LS2000_Attached_D := NDC8.UserDefined.Integer32_58_LS2000_Attached_D + 1;
	NDC8.UserDefined.Integer32_59_LS2000_Attached_H := 0;
end_if;

TravelDistanceSamplingTimer(IN:= TRUE, PT:=t#5s);

if TravelDistanceSamplingTimer.Q then
	if abs(NDC8.DCD_5.DriveEncDist - LastEncoderDistance) > 60000 then
		CurrentEncoderDistance := 65530 - abs(NDC8.DCD_5.DriveEncDist - LastEncoderDistance);
	else
		CurrentEncoderDistance := abs(NDC8.DCD_5.DriveEncDist - LastEncoderDistance);
	end_if;

	CurrentEncoderDistance := CurrentEncoderDistance / 10;

	NDC8.UserDefined.Integer32_55_TravelDistance := NDC8.UserDefined.Integer32_55_TravelDistance + UINT_TO_DINT(CurrentEncoderDistance);

	if NDC8.UserDefined.Integer32_55_TravelDistance > 2100000000 then
		NDC8.UserDefined.Integer32_55_TravelDistance := 0;
	end_if;

	LastEncoderDistance := NDC8.DCD_5.DriveEncDist;
	TravelDistanceSamplingTimer(IN:= FALSE);
end_if;

(* Black Box Trigger
if g_FindSyncFlag = TRUE Then
	BootUpDelay(IN:= TRUE, PT:=t#180s);
End_if;

if g_ErrorCode <> 0 and NoErrorDelay.Q = TRUE then
	ErrorFlag := TRUE;
end_if;

ErrorTrigR(CLK:= ErrorFlag);

if ErrorTrigR.Q = TRUE then
	ErrorTrigFlag := TRUE;
end_if;

if BootUpDelay.Q = TRUE then
	if ErrorTrigFlag then
		NDC8.BlackBox.TrigReason:= 'Error Trigger';
		BlackBox();
		if BlackBox.Finished then
			ErrorTrigFlag := FALSE;
		end_if;
	end_if;
End_if;

if g_ErrorCode = 0 then
	NoErrorDelay(IN:= TRUE, PT:=t#60s);
else
	NoErrorDelay(IN:= FALSE);
end_if;
 *)

Display();

(*if HMI Set "Force Output" signal will overwrite in OPTX2*)
OPTX2();

DataUpdate();

END_PROGRAM
